UdIntms := SysTimeGetMs();
uiMsSecond := UDINT_TO_UINT((UdIntms - UdMsOffset)MOD 1000);   //计算微秒
DTimer_Str := UINT_TO_STRING(uiYear);
DTimer_Str := concat(DTimer_Str,'-');
DTimer_Str := concat(DTimer_Str,UINT_TO_STRING(uiMonth));
DTimer_Str := concat(DTimer_Str,'-');
DTimer_Str := concat(DTimer_Str,UINT_TO_STRING(uiDay));
DTimer_Str := concat(DTimer_Str,' ');
DTimer_Str := concat(DTimer_Str,UINT_TO_STRING(uiHour+8));
DTimer_Str := concat(DTimer_Str,':');
DTimer_Str := concat(DTimer_Str,UINT_TO_STRING(uiMinute));
DTimer_Str := concat(DTimer_Str,':');
DTimer_Str := concat(DTimer_Str,UINT_TO_STRING(uiSecond));
DTimer_Str := concat(DTimer_Str,':');
DTimer_Str := concat(DTimer_Str,UINT_TO_STRING(uiMsSecond));
DTimer_Str := concat(DTimer_Str,'    ');

log_Str := concat(Log_Data,'$R');
F_HANDL :=SysFileOpen(szFile:= Filename, am:=ACCESS_MODE.AM_APPEND, pResult:= ADR(F_err));  //打开文件
SysFileGetPos(hFile:= F_HANDL , pulPos:= ADR(F_pos));		//获取文件位置
SysFileSetPos(hFile:= F_HANDL, ulOffset:= F_pos);
SysFileWrite(hFile:=F_HANDL , pbyBuffer:= ADR(DTimer_Str) , ulSize:= SysStrLen(DTimer_Str) , pResult:= ADR(F_err));		// 写入时间
SysFileWrite(hFile:=F_HANDL , pbyBuffer:= ADR(log_Str) , ulSize:= SysStrLen(log_Str) , pResult:= ADR(F_err));		// 写入数据
SysFileClose(hFile:=F_HANDL );

Out_log := concat(DTimer_Str,log_Str);

END_FUNCTION_BLOCK

// Device/Application/modbus/getObjIndexC
FUNCTION_BLOCK FINAL getObjIndexC
VAR_INPUT
	iAdr	:UINT;
	iBit	:UINT;
END_VAR
VAR_OUTPUT
	iO1		:USINT;
	iO2		:USINT;
END_VAR
VAR
END_VAR

//已知指令地址，获取对应比例阀索引及油缸编号索引
CASE iAdr OF
	10,13:
		CASE iBit OF
			1:		iO1:=3;iO2:=1;//Q01-04
			2:		iO1:=4;iO2:=1;//Q05-08
			3:		iO1:=5;iO2:=1;//Q09-12
			4:		iO1:=6;iO2:=1;//Q13-14
			5:		iO1:=6;iO2:=2;//Q15
			6:		iO1:=7;iO2:=4;//Q17-21
			7:		iO1:=7;iO2:=5;//Q22-26
			8:		iO1:=1;iO2:=5;//Q28
			9:		iO1:=1;iO2:=4;//Q29-30
			ELSE	iO1:=0;iO2:=0;	
		END_CASE

	11,14:
		CASE iBit OF
			0:		iO1:=1;iO2:=3;//L00
			ELSE	iO1:=0;iO2:=0;
		END_CASE	
	
	12,15:
		CASE iBit OF
			0:		iO1:=1;iO2:=6;//L01
			1:		iO1:=2;iO2:=1;//L02-04
			2:		iO1:=2;iO2:=2;//L05
			3:		iO1:=2;iO2:=3;//L06-08
			4:		iO1:=2;iO2:=4;//L09
			5:		iO1:=2;iO2:=5;//L10-12
			6:		iO1:=6;iO2:=4;//L13
			7:		iO1:=6;iO2:=3;//L14-15
			8:		iO1:=6;iO2:=5;//L16
			9:		iO1:=7;iO2:=6;//L17
			10:		iO1:=7;iO2:=1;//L18-21
			11:		iO1:=7;iO2:=2;//L22
			12:		iO1:=7;iO2:=3;//L23-26
			13:		iO1:=7;iO2:=7;//L27
			14:		iO1:=1;iO2:=1;//L28
			15:		iO1:=1;iO2:=2;//L29-30
			ELSE	iO1:=0;iO2:=0;
		END_CASE	
	ELSE
		iO1:=0;iO2:=0;	
END_CASE

END_FUNCTION_BLOCK

// Device/Application/modbus/getColumnStr
FUNCTION_BLOCK FINAL getColumnStr
VAR_INPUT
	iI1		:UINT;
	iI2		:UINT;
END_VAR
VAR_OUTPUT
	strO	:STRING;
END_VAR
VAR
END_VAR

CASE iI1 OF
	1:
	CASE iI2 OF
		1:strO:='E28L1-E28L2';
		2:strO:='E29L-E30L';
		3:strO:='E00L';
		4:strO:='E29Q-E30Q';
		5:strO:='E28Q';
		6:strO:='E01L';
	END_CASE
	2:
	CASE iI2 OF
		1:strO:='E02L-E04L';
		2:strO:='E05L';
		3:strO:='E06L-E08L';
		4:strO:='E09L';
		5:strO:='E10L-E12L';
	END_CASE
	3:strO:='E01Q1-E04Q2';
	4:strO:='E05Q1-E08Q2';
	5:strO:='E09Q1-E12Q2';
	6:
	CASE iI2 OF
		1:strO:='E13Q-E14Q';
		2:strO:='E15Q';
		3:strO:='E14L-E15L';
		4:strO:='E13L';
		5:strO:='E16L1-E16L2';

	END_CASE
	7:
	CASE iI2 OF
		1:strO:='E18L-E21L';
		2:strO:='E22L';
		3:strO:='E23L-E26L';
		4:strO:='E17Q-E21Q';
		5:strO:='E22Q-E26Q';
		6:strO:='E17L1-E17L2';
		7:strO:='E27L1-E27L2';
	END_CASE	
END_CASE

END_FUNCTION_BLOCK

// Device/Application/modbus/getObjIndexE
FUNCTION_BLOCK getObjIndexE
VAR_INPUT
	iI1:INT;
	iI2:INT;
END_VAR
VAR_OUTPUT
	iAdr:USINT;
END_VAR
VAR
	
END_VAR

//Modbus中，输入油缸编号索引，返回用于地址用于写入伸出状态是否到位
CASE iI1 OF
	1:
		CASE iI2 OF
			1:iAdr:=139;//L28
			2:iAdr:=140;//L29-L30
			3:iAdr:=124;//L00
			4:iAdr:=119;//Q29-Q30
			5:iAdr:=118;//Q28
			6:iAdr:=125;//L01
		END_CASE
	2:
		CASE iI2 OF
			1:iAdr:=126;//L02-04
			2:iAdr:=127;//L05
			3:iAdr:=128;//L06-08
			4:iAdr:=129;//L09
			5:iAdr:=130;//L10-12
		END_CASE
	3:iAdr:=111;//Q01-04
	4:iAdr:=112;//Q05-08
	5:iAdr:=113;//Q09-12
	6:
		CASE iI2 OF
			1:iAdr:=114;//Q13-14
			2:iAdr:=115;//Q15
			3:iAdr:=132;//L14-15
			4:iAdr:=131;//L13
			5:iAdr:=133;//L16
		END_CASE
	7:
		CASE iI2 OF
			1:iAdr:=135;//L18-21
			2:iAdr:=136;//L22
			3:iAdr:=137;//L23-26
			4:iAdr:=116;//Q17-21
			5:iAdr:=117;//Q22-26
			6:iAdr:=134;//L17
			7:iAdr:=138;//L27
		END_CASE

ELSE	
	iAdr:=0;
END_CASE

END_FUNCTION_BLOCK

// Device/Application/modbus/getObjIndexR
FUNCTION_BLOCK getObjIndexR
VAR_INPUT
	iI1:INT;
	iI2:INT;
END_VAR
VAR_OUTPUT
	iAdr:USINT;
END_VAR
VAR
	
END_VAR

//Modbus中，输入油缸编号索引，返回用于地址用于写入缩回状态是否到位
CASE iI1 OF
	1:		
		CASE iI2 OF	
			1:iAdr:=170;//L28
			2:iAdr:=171;//L29-30
			3:iAdr:=155;//L00
			4:iAdr:=150;//Q29-30
			5:iAdr:=149;//Q28
			6:iAdr:=156;//L01
		END_CASE	
	2:		
		CASE iI2 OF	
			1:iAdr:=157;//L02-04
			2:iAdr:=158;//L05
			3:iAdr:=159;//L06-08
			4:iAdr:=160;//L09
			5:iAdr:=161;//L10-12
		END_CASE	
	3:iAdr:=142;//Q01-04		
	4:iAdr:=143;//Q05-08		
	5:iAdr:=144;//Q09-12		
	6:		
		CASE iI2 OF	
			1:iAdr:=145;//Q13-14
			2:iAdr:=146;//Q15
			3:iAdr:=163;//L14-15
			4:iAdr:=162;//L13
			5:iAdr:=164;//L16
		END_CASE	
	7:		
		CASE iI2 OF	
			1:iAdr:=166;//L18-21
			2:iAdr:=167;//L22
			3:iAdr:=168;//L23-26
			4:iAdr:=147;//Q17-21
			5:iAdr:=148;//Q22-26
			6:iAdr:=165;//L17
			7:iAdr:=169;//L27
		END_CASE	


ELSE	
	iAdr:=0;
END_CASE

END_FUNCTION_BLOCK

// Device/Application/rail_ceiling/positionRecord
PROGRAM positionRecord
VAR
	arrPosVal			:ARRAY[1..200] OF UINT;
	fbDatSav			:DatSave;
	iT1					:UINT;
	iT2					:UINT;
	iNum				:UINT;
END_VAR
VAR CONSTANT
	aOil	:ARRAY [1..7] OF UINT :=[9,11,8,8,8,8,23];		
END_VAR

iNum:=1;
FOR iT1:=1 TO 7 DO
	FOR iT2:=1 TO aOil[iT1] DO
		arrPosVal[iNum]:=REAL_TO_UINT(gImple.PV_GroupTi.arrPV[iT1].sNum[iT2].posVal.Current);
		iNum:=iNum+1;
	END_FOR
END_FOR
fbDatSav(Data_Arry:=arrPosVal , Num:= 75 , FilePath:= 'D:/DataSave', cycle:= T#7200S);

END_PROGRAM

// Device/Application/public_datum/datarecord/datSave
FUNCTION_BLOCK datSave
VAR_INPUT
	Data_Arry	: ARRAY[1..200] OF UINT;	// 数据输入 一次最大可以写入200个数据
	Num			: UINT;						// 存储数据个数
	FilePath 	: STRING := 'C:/DataSave'; 	// 存储文件夹
	cycle		: TIME;						// 更新一个文件夹时间
END_VAR
VAR_OUTPUT
END_VAR
VAR
	datetime	: DATE_AND_TIME;
	uiYear 		: UINT; 
    uiMonth 	: UINT; 
    uiDay 		: UINT; 
    uiHour 		: UINT; 
    uiMinute 	: UINT; 
    uiSecond 	: UINT;	
	uiMsSecond	: UINT;
	Last_S		: UINT:=100;
	UdMsOffset  : UDINT;
	UdIntms 	: UDINT;
	DTimer_Arry : ARRAY[1..7] OF UINT;
END_VAR
VAR
	File_Init	: BOOL :=TRUE;
	Frame_Cnt	: LINT;
	Data_Save_Init :BOOL:=TRUE;
	New_File_Ton: TON;
	Filename	: STRING;
	F_HANDL		: DWORD;
	F_err		: DWORD;
	F_pos		: DWORD;
END_VAR

datetime:=GetDateTime();   //获取时间
DTU.DTSplit(
		dtDateAndTime:= datetime, 
		puiYear:= ADR(uiYear), 
		puiMonth:=  ADR(uiMonth), 
		puiDay:=  ADR(uiDay), 
		puiHour:=  ADR(uiHour), 
		puiMinute:=  ADR(uiMinute), 
		puiSecond:= ADR(uiSecond) );

IF  Data_Save_Init THEN			//数据存储初始化
	IF uiSecond = Last_S +1 OR  uiSecond = Last_S -59 THEN
		UdMsOffset := SysTimeGetMs();
		Last_S :=  uiSecond;
	ELSE
		Last_S :=  uiSecond;
		RETURN;
	END_IF
    Data_Save_Init := FALSE;
END_IF

IF 	File_Init  THEN          //创建文件
	Filename := FilePath;
	Filename := concat(Filename,'/');
	Filename := concat(Filename,UINT_TO_STRING(uiYear));
	Filename := concat(Filename,'_');
	Filename := concat(Filename,UINT_TO_STRING(uiMonth));
	Filename := concat(Filename,'_');
	Filename := concat(Filename,UINT_TO_STRING(uiDay));
	Filename := concat(Filename,'_');
	Filename := concat(Filename,UINT_TO_STRING(uiHour+8));
 	Filename := concat(Filename,'_');
	Filename := concat(Filename,UINT_TO_STRING(uiMinute));
	Filename := concat(Filename,'_');
	Filename := concat(Filename,UINT_TO_STRING(uiSecond));
    Filename := concat(Filename,'_Data.bin');
	Frame_Cnt := 0;
	F_HANDL :=SysFileOpen(szFile:= Filename, am:=ACCESS_MODE.AM_WRITE, pResult:= ADR(F_err));  //创建新文件
	SysFileClose(hFile:=F_HANDL );
	File_Init := FALSE;
	New_File_Ton(IN:= FALSE , PT:= cycle, Q=> , ET=> );  //复位
END_IF

New_File_Ton(IN:= TRUE , PT:= cycle, Q=> , ET=> );			//4小时创建一个新文件
IF New_File_Ton.Q THEN
	File_Init := TRUE;	
END_IF



UdIntms := SysTimeGetMs();
DTimer_Arry[1] := uiYear;
DTimer_Arry[2] := uiMonth;
DTimer_Arry[3] := uiDay;
DTimer_Arry[4] := uiHour+8;
DTimer_Arry[5] := uiMinute;
DTimer_Arry[6] := uiSecond;
DTimer_Arry[7] := UDINT_TO_UINT((UdIntms - UdMsOffset)MOD 1000);

Frame_Cnt := Frame_Cnt + 1;    	//帧计数增加

F_HANDL :=SysFileOpen(szFile:= Filename, am:=ACCESS_MODE.AM_APPEND, pResult:= ADR(F_err));  //打开文件
SysFileGetPos(hFile:= F_HANDL , pulPos:= ADR(F_pos));		//获取文件位置
SysFileSetPos(hFile:= F_HANDL, ulOffset:= 0);	//设置帧位置
SysFileWrite(hFile:=F_HANDL , pbyBuffer:= ADR(Frame_Cnt) , ulSize:= SIZEOF(Frame_Cnt) , pResult:= ADR(F_err));    //修改总帧数
IF F_pos <> 0 THEN		//不是新文件，设置写入位置
	SysFileSetPos(hFile:= F_HANDL, ulOffset:= F_pos);
END_IF
SysFileWrite(hFile:=F_HANDL , pbyBuffer:= ADR(DTimer_Arry) , ulSize:= SIZEOF(DTimer_Arry) , pResult:= ADR(F_err));  // 保存时间
SysFileWrite(hFile:=F_HANDL , pbyBuffer:= ADR(Data_Arry) , ulSize:= SIZEOF(UINT)*Num , pResult:= ADR(F_err));		// 保存数据
SysFileClose(hFile:=F_HANDL );

END_FUNCTION_BLOCK

// Device/Application/can/canRx
PROGRAM canRx
VAR
		T_CNT   :UINT;
END_VAR

T_CNT := T_CNT+1;
IF  T_CNT > 1000 THEN
	 T_CNT := 1;
END_IF


swmc_C05_Rx(T_CNT,ADR(gImple.hydraPresStation),ADR(gImple.PV_GroupTi));
swmc_C06_Rx(T_CNT,ADR(gImple.hydraPresStation),ADR(gImple.PV_GroupTi));
swmc_C12_Rx(T_CNT,ADR(gImple.PV_GroupTi));

END_PROGRAM

// Device/Application/can/swmc_C05_Rx
FUNCTION swmc_C05_Rx : BOOL
VAR_INPUT
	CNT				: UINT;
	psYyz			: POINTER TO YyStation;
	psPVTi			: POINTER TO propValveModule_Ti;

END_VAR
VAR
	frame	 	    : Can_baseframe;
	COB_ID			: UINT;
	I				: UINT;
	Pre				: UINT;
	pos				: WORD;
END_VAR

IF gCan.C5RxMsg.RxCounter <>  gCan.C5RxCounter THEN    //接收到新的数据

	FOR  I := 1 TO  gCan.C5RxMsg.NoOfRxMessages DO
		frame :=CAN_Read_Data_SWMC(5,I);
		COB_ID :=	frame.id;    //获取ID
		CASE COB_ID OF     //根据ID解析协议
		
		//C5-0x350
			16#350://接收C5送来的数据
				pos := BYTE_TO_WORD(frame.data[1]) OR SHL(BYTE_TO_WORD(frame.data[2]),8);  	
				psPVTi^.arrPV[3].sNum[1].posVal.Current:= pos*0.1;
				pos := BYTE_TO_WORD(frame.data[3]) OR SHL(BYTE_TO_WORD(frame.data[4]),8);  
				psPVTi^.arrPV[3].sNum[2].posVal.Current:= pos*0.1;	
				pos := BYTE_TO_WORD(frame.data[5]) OR SHL(BYTE_TO_WORD(frame.data[6]),8);  
				psPVTi^.arrPV[3].sNum[3].posVal.Current:= pos*0.1;	
				pos := BYTE_TO_WORD(frame.data[7]) OR SHL(BYTE_TO_WORD(frame.data[8]),8);  	
				psPVTi^.arrPV[3].sNum[4].posVal.Current:= pos*0.1;
			
			//C5-0x351
			16#351://接收C5送来的数据
				pos := BYTE_TO_WORD(frame.data[1]) OR SHL(BYTE_TO_WORD(frame.data[2]),8);  	
				psPVTi^.arrPV[3].sNum[5].posVal.Current:= pos*0.1;	
				pos := BYTE_TO_WORD(frame.data[3]) OR SHL(BYTE_TO_WORD(frame.data[4]),8);  	
				psPVTi^.arrPV[3].sNum[6].posVal.Current:= pos*0.1;	
				pos := BYTE_TO_WORD(frame.data[5]) OR SHL(BYTE_TO_WORD(frame.data[6]),8);  	
				psPVTi^.arrPV[3].sNum[7].posVal.Current:= pos*0.1;	
				pos := BYTE_TO_WORD(frame.data[7]) OR SHL(BYTE_TO_WORD(frame.data[8]),8);  	
				psPVTi^.arrPV[3].sNum[8].posVal.Current:= pos*0.1;
			
			//C5-0x352
			16#352://接收C5送来的数据
			pos := BYTE_TO_WORD(frame.data[1]) OR SHL(BYTE_TO_WORD(frame.data[2]),8);  	
				psPVTi^.arrPV[4].sNum[1].posVal.Current:= pos*0.1;	
				pos := BYTE_TO_WORD(frame.data[3]) OR SHL(BYTE_TO_WORD(frame.data[4]),8);  	
				psPVTi^.arrPV[4].sNum[2].posVal.Current:= pos*0.1;		
				pos := BYTE_TO_WORD(frame.data[5]) OR SHL(BYTE_TO_WORD(frame.data[6]),8);  	
				psPVTi^.arrPV[4].sNum[3].posVal.Current:= pos*0.1;		
				pos := BYTE_TO_WORD(frame.data[7]) OR SHL(BYTE_TO_WORD(frame.data[8]),8);  	
				psPVTi^.arrPV[4].sNum[4].posVal.Current:= pos*0.1;	
			
			//C5-0x353
			16#353://接收C5送来的数据
				pos := BYTE_TO_WORD(frame.data[1]) OR SHL(BYTE_TO_WORD(frame.data[2]),8);  	
				psPVTi^.arrPV[4].sNum[5].posVal.Current:= pos*0.1;		
				pos := BYTE_TO_WORD(frame.data[3]) OR SHL(BYTE_TO_WORD(frame.data[4]),8);  	
				psPVTi^.arrPV[4].sNum[6].posVal.Current:= pos*0.1;		
				pos := BYTE_TO_WORD(frame.data[5]) OR SHL(BYTE_TO_WORD(frame.data[6]),8);  	
				psPVTi^.arrPV[4].sNum[7].posVal.Current:= pos*0.1;		
				pos := BYTE_TO_WORD(frame.data[7]) OR SHL(BYTE_TO_WORD(frame.data[8]),8);  	
				psPVTi^.arrPV[4].sNum[8].posVal.Current:= pos*0.1;	
			
			//C5-0x354
			16#354://接收C5送来的数据
			pos := BYTE_TO_WORD(frame.data[1]) OR SHL(BYTE_TO_WORD(frame.data[2]),8);  	
				psPVTi^.arrPV[5].sNum[1].posVal.Current:= pos*0.1;		
				pos := BYTE_TO_WORD(frame.data[3]) OR SHL(BYTE_TO_WORD(frame.data[4]),8);  	
				psPVTi^.arrPV[5].sNum[2].posVal.Current:= pos*0.1;		
				pos := BYTE_TO_WORD(frame.data[5]) OR SHL(BYTE_TO_WORD(frame.data[6]),8);  	
				psPVTi^.arrPV[5].sNum[3].posVal.Current:= pos*0.1;		
				pos := BYTE_TO_WORD(frame.data[7]) OR SHL(BYTE_TO_WORD(frame.data[8]),8);  	
				psPVTi^.arrPV[5].sNum[4].posVal.Current:= pos*0.1;	
			
			//C5-0x355
			16#355://接收C5送来的数据
			pos := BYTE_TO_WORD(frame.data[1]) OR SHL(BYTE_TO_WORD(frame.data[2]),8);  	
				psPVTi^.arrPV[5].sNum[5].posVal.Current:= pos*0.1;		
				pos := BYTE_TO_WORD(frame.data[3]) OR SHL(BYTE_TO_WORD(frame.data[4]),8);  	
				psPVTi^.arrPV[5].sNum[6].posVal.Current:= pos*0.1;		
				pos := BYTE_TO_WORD(frame.data[5]) OR SHL(BYTE_TO_WORD(frame.data[6]),8);  	
				psPVTi^.arrPV[5].sNum[7].posVal.Current:= pos*0.1;		
				pos := BYTE_TO_WORD(frame.data[7]) OR SHL(BYTE_TO_WORD(frame.data[8]),8);  	
				psPVTi^.arrPV[5].sNum[8].posVal.Current:= pos*0.1;	
			

	
			//C5-0x356
			16#356:           //接收C5送来的数据
			(*
				Pre :=BYTE_TO_WORD(frame.data[1]) OR SHL(BYTE_TO_WORD(frame.data[2]),8);
				psYyz^.Status.pressureV10:= 	(Pre-4000)/16000.0*400;	
				Pre :=BYTE_TO_WORD(frame.data[3]) OR SHL(BYTE_TO_WORD(frame.data[4]),8);
				psYyz^.Status.pressureV11:= 	(Pre-4000)/16000.0*400;	
			*)
			
	
		END_CASE
	END_FOR
	gCan.C5RxCounter := gCan.C5RxMsg.RxCounter ;
END_IF

END_FUNCTION

// Device/Application/can/CAN_Read_Data_SWMC
FUNCTION CAN_Read_Data_SWMC : Can_baseframe
VAR_INPUT
	SWMC_ID	 :UINT;		//接收SWMC控制ID
	I	 	 :UINT;      //接收缓冲区域
END_VAR
VAR
	frame :Can_baseframe;
END_VAR

CASE  SWMC_ID OF

	5:                       //SWMC-C5
		frame.id 	:= (gCan.C5RxMsg.RXMsg[I].RxMsg_CobId-8)/32;
		frame.data 	:= gCan.C5RxMsg.RXMsg[I].RxMsg_Byte;
				
	6:                       //SWMC-C6
		frame.id 	:= (gCan.C6RxMsg.RXMsg[I].RxMsg_CobId-8)/32;
		frame.data 	:= gCan.C6RxMsg.RXMsg[I].RxMsg_Byte;

	12:						//SWMC-C12
		frame.id 	:= (gCan.C12RxMsg.RXMsg[I].RxMsg_CobId-8)/32;
		frame.data 	:= gCan.C12RxMsg.RXMsg[I].RxMsg_Byte;	
		
	ELSE				//Other
		frame.id := 0;
		frame.data[1] := 0;
		frame.data[2] := 0;
		frame.data[3] := 0;
		frame.data[4] := 0;
		frame.data[5] := 0;
		frame.data[6] := 0;
		frame.data[7] := 0;
		frame.data[8] := 0;
END_CASE
Can_Read_data_SWMC := frame;

END_FUNCTION

// Device/Application/can/swmc_C06_Rx
FUNCTION swmc_C06_Rx : BOOL
VAR_INPUT
	CNT				: UINT;
	psYyz			: POINTER TO YyStation;
	psPVTi			: POINTER TO propValveModule_Ti;

END_VAR
VAR
	frame	 	    : Can_baseframe;
	COB_ID			: UINT;
	I				: UINT;
	Pre				: UINT;
	pos				: WORD;
END_VAR

IF gCan.C6RxMsg.RxCounter <>  gCan.C6RxCounter THEN    //接收到新的数据

	FOR  I := 1 TO  gCan.C6RxMsg.NoOfRxMessages DO
		frame :=CAN_Read_Data_SWMC(6,I);
		COB_ID :=	frame.id;    //获取ID
		CASE COB_ID OF     //根据ID解析协议
	
		
			//C6-0x360
			16#360:           //接收C6送来的数据
				pos:=BYTE_TO_WORD(frame.data[1]) OR SHL(BYTE_TO_WORD(frame.data[2]),8);
				psPVTi^.arrPV[1].sNum[3].posVal.Current:=pos*0.1;
				pos:=BYTE_TO_WORD(frame.data[3]) OR SHL(BYTE_TO_WORD(frame.data[4]),8);
				psPVTi^.arrPV[1].sNum[4].posVal.Current:=pos*0.1;
				pos:=BYTE_TO_WORD(frame.data[5]) OR SHL(BYTE_TO_WORD(frame.data[6]),8);
				psPVTi^.arrPV[1].sNum[9].posVal.Current:=pos*0.1;
				pos:=BYTE_TO_WORD(frame.data[7]) OR SHL(BYTE_TO_WORD(frame.data[8]),8);
				psPVTi^.arrPV[1].sNum[5].posVal.Current:=pos*0.1;
			

			//C6-0x361
			16#361:           //接收C6送来的数据
				pos:=BYTE_TO_WORD(frame.data[1]) OR SHL(BYTE_TO_WORD(frame.data[2]),8);
				psPVTi^.arrPV[1].sNum[8].posVal.Current:=pos*0.1;
				pos:=BYTE_TO_WORD(frame.data[3]) OR SHL(BYTE_TO_WORD(frame.data[4]),8);
				psPVTi^.arrPV[1].sNum[6].posVal.Current:=pos*0.1;
				pos:=BYTE_TO_WORD(frame.data[5]) OR SHL(BYTE_TO_WORD(frame.data[6]),8);
				psPVTi^.arrPV[1].sNum[7].posVal.Current:=pos*0.1;
				pos:=BYTE_TO_WORD(frame.data[7]) OR SHL(BYTE_TO_WORD(frame.data[8]),8);
				psPVTi^.arrPV[2].sNum[1].posVal.Current:=pos*0.1;
			//C6-0x362
			16#362:           //接收C6送来的数据
				pos:=BYTE_TO_WORD(frame.data[1]) OR SHL(BYTE_TO_WORD(frame.data[2]),8);
				psPVTi^.arrPV[2].sNum[2].posVal.Current:=pos*0.1;
				pos:=BYTE_TO_WORD(frame.data[3]) OR SHL(BYTE_TO_WORD(frame.data[4]),8);
				psPVTi^.arrPV[2].sNum[3].posVal.Current:=pos*0.1;
				pos:=BYTE_TO_WORD(frame.data[5]) OR SHL(BYTE_TO_WORD(frame.data[6]),8);
				psPVTi^.arrPV[2].sNum[4].posVal.Current:=pos*0.1;
				pos:=BYTE_TO_WORD(frame.data[7]) OR SHL(BYTE_TO_WORD(frame.data[8]),8);
				psPVTi^.arrPV[2].sNum[5].posVal.Current:=pos*0.1;
			//C6-0x363
			16#363:           //接收C6送来的数据
				pos:=BYTE_TO_WORD(frame.data[1]) OR SHL(BYTE_TO_WORD(frame.data[2]),8);
				psPVTi^.arrPV[2].sNum[6].posVal.Current:=pos*0.1;
				pos:=BYTE_TO_WORD(frame.data[3]) OR SHL(BYTE_TO_WORD(frame.data[4]),8);
				psPVTi^.arrPV[2].sNum[7].posVal.Current:=pos*0.1;
				pos:=BYTE_TO_WORD(frame.data[5]) OR SHL(BYTE_TO_WORD(frame.data[6]),8);
				psPVTi^.arrPV[2].sNum[8].posVal.Current:=pos*0.1;
				pos:=BYTE_TO_WORD(frame.data[7]) OR SHL(BYTE_TO_WORD(frame.data[8]),8);
				psPVTi^.arrPV[2].sNum[9].posVal.Current:=pos*0.1;
			//C6-0x364
			16#364:           //接收C6送来的数据
				pos:=BYTE_TO_WORD(frame.data[1]) OR SHL(BYTE_TO_WORD(frame.data[2]),8);
				psPVTi^.arrPV[2].sNum[10].posVal.Current:=pos*0.1;
				pos:=BYTE_TO_WORD(frame.data[3]) OR SHL(BYTE_TO_WORD(frame.data[4]),8);
				psPVTi^.arrPV[2].sNum[11].posVal.Current:=pos*0.1;
				pos:=BYTE_TO_WORD(frame.data[5]) OR SHL(BYTE_TO_WORD(frame.data[6]),8);
				psPVTi^.arrPV[6].sNum[6].posVal.Current:=pos*0.1;
				pos:=BYTE_TO_WORD(frame.data[7]) OR SHL(BYTE_TO_WORD(frame.data[8]),8);
				psPVTi^.arrPV[6].sNum[4].posVal.Current:=pos*0.1;
			//C6-0x365
			16#365:           //接收C6送来的数据
				pos:=BYTE_TO_WORD(frame.data[1]) OR SHL(BYTE_TO_WORD(frame.data[2]),8);
				psPVTi^.arrPV[6].sNum[5].posVal.Current:=pos*0.1;
				pos:=BYTE_TO_WORD(frame.data[3]) OR SHL(BYTE_TO_WORD(frame.data[4]),8);
				psPVTi^.arrPV[6].sNum[1].posVal.Current:=pos*0.1;
				pos:=BYTE_TO_WORD(frame.data[5]) OR SHL(BYTE_TO_WORD(frame.data[6]),8);
				psPVTi^.arrPV[6].sNum[2].posVal.Current:=pos*0.1;
				pos:=BYTE_TO_WORD(frame.data[7]) OR SHL(BYTE_TO_WORD(frame.data[8]),8);
				psPVTi^.arrPV[6].sNum[3].posVal.Current:=pos*0.1;
				
		
			//C6-0x366
			16#366:           //接收C6送来的数据
				//Pre :=BYTE_TO_WORD(frame.data[1]) OR SHL(BYTE_TO_WORD(frame.data[2]),8);
	 			//psYyz^.Status.pressureV8:= 	(Pre-4000)/16000.0*400;	
				//Pre :=BYTE_TO_WORD(frame.data[3]) OR SHL(BYTE_TO_WORD(frame.data[4]),8);
	 			//psYyz^.Status.pressureV9:= 	(Pre-4000)/16000.0*400;	
				pos	:=BYTE_TO_WORD(frame.data[5]) OR SHL(BYTE_TO_WORD(frame.data[6]),8);
				psPVTi^.arrAddtion[1].sPlateStatus.sSensor.Current:=pos*0.1;
				pos	:=BYTE_TO_WORD(frame.data[7]) OR SHL(BYTE_TO_WORD(frame.data[8]),8);
				psPVTi^.arrAddtion[2].sPlateStatus.sSensor.Current:=pos*0.1;
				
		END_CASE
	END_FOR
	gCan.C6RxCounter := gCan.C6RxMsg.RxCounter ;
END_IF

END_FUNCTION

// Device/Application/can/swmc_C12_Rx
FUNCTION swmc_C12_Rx : BOOL
VAR_INPUT
	CNT				: UINT;
	psPVTi			: POINTER TO propValveModule_Ti;
END_VAR
VAR
	frame	 	    : Can_baseframe;
	COB_ID			: UINT;
	I				: UINT;
	Pre				: UINT;
	pos				: WORD;
END_VAR

IF gCan.C12RxMsg.RxCounter <>  gCan.C12RxCounter THEN    //接收到新的数据

	FOR  I := 1 TO  gCan.C12RxMsg.NoOfRxMessages DO
		frame :=CAN_Read_Data_SWMC(12,I);
		COB_ID :=	frame.id;    //获取ID
		CASE COB_ID OF     //根据ID解析协议
		
		
			//C12-0x3C0
			16#3C0:           //接收C12送来的数据
				pos := BYTE_TO_WORD(frame.data[ 1 ]) OR SHL(BYTE_TO_WORD(frame.data[ 2 ]),8);  	
				psPVTi^.arrPV[ 6 ].sNum[ 7 ].posVal.Current:= pos*0.1;	
				pos := BYTE_TO_WORD(frame.data[ 3 ]) OR SHL(BYTE_TO_WORD(frame.data[ 4 ]),8);  
				psPVTi^.arrPV[ 6 ].sNum[ 8 ].posVal.Current:= pos*0.1;		
				pos := BYTE_TO_WORD(frame.data[ 5 ]) OR SHL(BYTE_TO_WORD(frame.data[ 6 ]),8);  
				psPVTi^.arrPV[ 7 ].sNum[ 20 ].posVal.Current:= pos*0.1;	
				pos := BYTE_TO_WORD(frame.data[ 7 ]) OR SHL(BYTE_TO_WORD(frame.data[ 8 ]),8);  	
				psPVTi^.arrPV[ 7 ].sNum[ 21 ].posVal.Current:= pos*0.1;

			//C6-0x3C1
			16#3C1:           //接收C12送来的数据
				pos := BYTE_TO_WORD(frame.data[ 1 ]) OR SHL(BYTE_TO_WORD(frame.data[ 2 ]),8);  	
				psPVTi^.arrPV[ 7 ].sNum[ 1 ].posVal.Current:= pos*0.1;	
				pos := BYTE_TO_WORD(frame.data[ 3 ]) OR SHL(BYTE_TO_WORD(frame.data[ 4 ]),8);  	
				psPVTi^.arrPV[ 7 ].sNum[ 2 ].posVal.Current:= pos*0.1;	
				pos := BYTE_TO_WORD(frame.data[ 5 ]) OR SHL(BYTE_TO_WORD(frame.data[ 6 ]),8);  	
				psPVTi^.arrPV[ 7 ].sNum[ 3 ].posVal.Current:= pos*0.1;	
				pos := BYTE_TO_WORD(frame.data[ 7 ]) OR SHL(BYTE_TO_WORD(frame.data[ 8 ]),8);  	
				psPVTi^.arrPV[ 7 ].sNum[ 4 ].posVal.Current:= pos*0.1;
			//C6-0x3C2
			16#3C2:           //接收C12送来的数据
				pos := BYTE_TO_WORD(frame.data[ 1 ]) OR SHL(BYTE_TO_WORD(frame.data[ 2 ]),8);  	
				psPVTi^.arrPV[ 7 ].sNum[ 5 ].posVal.Current:= pos*0.1;	
				pos := BYTE_TO_WORD(frame.data[ 3 ]) OR SHL(BYTE_TO_WORD(frame.data[ 4 ]),8);  	
				psPVTi^.arrPV[ 7 ].sNum[ 6 ].posVal.Current:= pos*0.1;		
				pos := BYTE_TO_WORD(frame.data[ 5 ]) OR SHL(BYTE_TO_WORD(frame.data[ 6 ]),8);  	
				psPVTi^.arrPV[ 7 ].sNum[ 7 ].posVal.Current:= pos*0.1;		
				pos := BYTE_TO_WORD(frame.data[ 7 ]) OR SHL(BYTE_TO_WORD(frame.data[ 8 ]),8);  	
				psPVTi^.arrPV[ 7 ].sNum[ 8 ].posVal.Current:= pos*0.1;	
			//C6-0x3C3
			16#3C3:           //接收C12送来的数据
				pos := BYTE_TO_WORD(frame.data[ 1 ]) OR SHL(BYTE_TO_WORD(frame.data[ 2 ]),8);  	
				psPVTi^.arrPV[ 7 ].sNum[ 9 ].posVal.Current:= pos*0.1;		
				pos := BYTE_TO_WORD(frame.data[ 3 ]) OR SHL(BYTE_TO_WORD(frame.data[ 4 ]),8);  	
				psPVTi^.arrPV[ 7 ].sNum[ 22 ].posVal.Current:= pos*0.1;		
				pos := BYTE_TO_WORD(frame.data[ 5 ]) OR SHL(BYTE_TO_WORD(frame.data[ 6 ]),8);  	
				psPVTi^.arrPV[7 ].sNum[ 23 ].posVal.Current:= pos*0.1;		
				pos := BYTE_TO_WORD(frame.data[ 7 ]) OR SHL(BYTE_TO_WORD(frame.data[ 8 ]),8);  	
				psPVTi^.arrPV[ 1 ].sNum[ 1 ].posVal.Current:= pos*0.1;	
			//C6-0x3C4
			16#3C4:           //接收C12送来的数据
				pos := BYTE_TO_WORD(frame.data[ 1 ]) OR SHL(BYTE_TO_WORD(frame.data[ 2 ]),8);  	
				psPVTi^.arrPV[ 1 ].sNum[ 2 ].posVal.Current:= pos*0.1;		
				pos := BYTE_TO_WORD(frame.data[ 3 ]) OR SHL(BYTE_TO_WORD(frame.data[ 4 ]),8);  	
				psPVTi^.arrPV[ 7 ].sNum[ 10 ].posVal.Current:= pos*0.1;		
				pos := BYTE_TO_WORD(frame.data[ 5 ]) OR SHL(BYTE_TO_WORD(frame.data[ 6 ]),8);  	
				psPVTi^.arrPV[ 7 ].sNum[ 11 ].posVal.Current:= pos*0.1;		
				pos := BYTE_TO_WORD(frame.data[ 7 ]) OR SHL(BYTE_TO_WORD(frame.data[ 8 ]),8);  	
				psPVTi^.arrPV[7 ].sNum[ 12 ].posVal.Current:= pos*0.1;	
			//C6-0x3C5
			16#3C5:           //接收C12送来的数据
				pos := BYTE_TO_WORD(frame.data[ 1 ]) OR SHL(BYTE_TO_WORD(frame.data[ 2 ]),8);  	
				psPVTi^.arrPV[ 7 ].sNum[ 13 ].posVal.Current:= pos*0.1;		
				pos := BYTE_TO_WORD(frame.data[ 3 ]) OR SHL(BYTE_TO_WORD(frame.data[ 4 ]),8);  	
				psPVTi^.arrPV[ 7 ].sNum[ 14 ].posVal.Current:= pos*0.1;		
				pos := BYTE_TO_WORD(frame.data[ 5 ]) OR SHL(BYTE_TO_WORD(frame.data[ 6 ]),8);  	
				psPVTi^.arrPV[ 7 ].sNum[ 15 ].posVal.Current:= pos*0.1;		
				pos := BYTE_TO_WORD(frame.data[ 7 ]) OR SHL(BYTE_TO_WORD(frame.data[ 8 ]),8);  	
				psPVTi^.arrPV[ 7 ].sNum[ 16 ].posVal.Current:= pos*0.1;
			//C6-0x3C6
			16#3C6:           //接收C12送来的数据
				pos := BYTE_TO_WORD(frame.data[ 1 ]) OR SHL(BYTE_TO_WORD(frame.data[ 2 ]),8);  	
				psPVTi^.arrPV[ 7 ].sNum[ 17 ].posVal.Current:= pos*0.1;		
				pos := BYTE_TO_WORD(frame.data[ 3 ]) OR SHL(BYTE_TO_WORD(frame.data[ 4 ]),8);  	
				psPVTi^.arrPV[ 7 ].sNum[ 18 ].posVal.Current:= pos*0.1;		
				pos := BYTE_TO_WORD(frame.data[ 5 ]) OR SHL(BYTE_TO_WORD(frame.data[ 6 ]),8);  	
				psPVTi^.arrPV[ 7 ].sNum[ 19 ].posVal.Current:= pos*0.1;		
						
		
			
		END_CASE
	END_FOR
	gCan.C12RxCounter := gCan.C12RxMsg.RxCounter ;
END_IF

END_FUNCTION

// Device/Application/public_datum/otherContent/rail_floor/floorRailAct
PROGRAM floorRailAct
VAR
	bInitialize		:BOOL:=TRUE;
	iVD				:INT;
	iVD1			:INT;
END_VAR
VAR CONSTANT
	aNo		:ARRAY [1..7] OF INT :=[ 7, 5,1,1,1,5, 7];		//每个比例阀下开关阀的数量(天轨):arrMappingRealNumTiG
	aOil	:ARRAY [1..7] OF INT :=[12,11,8,8,8,8,23];		
END_VAR

IF bInitialize THEN	//初始化
	floorRailAct.initName();
	floorRailAct.initRange();
	bInitialize:=FALSE;
END_IF
statusDisplayDi();
CommandDeliverDi();

ACTION statusDisplayDi:
//初始化：名称显示，油缸位移范围赋值
initName();
initRange();


//	gUI.界面值<--gImple.传感器位置值;

//比例阀DTD1
FOR iVD	:=1 TO 12 DO
	gUI.DiG.arrPV[1].sNum[iVD].rPosition:=gImple.PV_GroupDi.arrPV[1].sNum[iVD].posVal.Current;
	gUI.DiG.arrPV[1].sNum[iVD].rPercent:=statusPercentCalcDi(ADR(gImple.PV_GroupDi),1,iVD);
	gUI.DiG.arrPV[1].sNum[iVD].strName:=gUI.DiG_NameInit.strName[1,iVD];
END_FOR

//比例阀DTD2
FOR iVD	:=1 TO 11 DO
	gUI.DiG.arrPV[2].sNum[iVD].rPosition:=gImple.PV_GroupDi.arrPV[2].sNum[iVD].posVal.Current;
	gUI.DiG.arrPV[2].sNum[iVD].rPercent:=statusPercentCalcDi(ADR(gImple.PV_GroupDi),2,iVD);
	gUI.DiG.arrPV[2].sNum[iVD].strName:=gUI.DiG_NameInit.strName[2,iVD];
END_FOR

//比例阀DTD345
FOR iVD	:=1 TO 8 DO

	gUI.DiG.arrPV[3].sNum[iVD].rPosition:=gImple.PV_GroupDi.arrPV[3].sNum[iVD].posVal.Current;
	gUI.DiG.arrPV[4].sNum[iVD].rPosition:=gImple.PV_GroupDi.arrPV[4].sNum[iVD].posVal.Current;
	gUI.DiG.arrPV[5].sNum[iVD].rPosition:=gImple.PV_GroupDi.arrPV[5].sNum[iVD].posVal.Current;
	
	gUI.DiG.arrPV[3].sNum[iVD].rPercent:=statusPercentCalcDi(ADR(gImple.PV_GroupDi),3,iVD);
	gUI.DiG.arrPV[4].sNum[iVD].rPercent:=statusPercentCalcDi(ADR(gImple.PV_GroupDi),4,iVD);
	gUI.DiG.arrPV[5].sNum[iVD].rPercent:=statusPercentCalcDi(ADR(gImple.PV_GroupDi),5,iVD);
	
	gUI.DiG.arrPV[3].sNum[iVD].strName:=gUI.DiG_NameInit.strName[3,iVD];
	gUI.DiG.arrPV[4].sNum[iVD].strName:=gUI.DiG_NameInit.strName[4,iVD];
	gUI.DiG.arrPV[5].sNum[iVD].strName:=gUI.DiG_NameInit.strName[5,iVD];
END_FOR

//比例阀DTD6
FOR iVD	:=1 TO 8 DO
	gUI.DiG.arrPV[6].sNum[iVD].rPosition:=gImple.PV_GroupDi.arrPV[6].sNum[iVD].posVal.Current;
	gUI.DiG.arrPV[6].sNum[iVD].rPercent:=statusPercentCalcDi(ADR(gImple.PV_GroupDi),6,iVD);
	gUI.DiG.arrPV[6].sNum[iVD].strName:=gUI.DiG_NameInit.strName[6,iVD];
END_FOR

//比例阀DTD7
FOR iVD	:=1 TO 23 DO
	gUI.DiG.arrPV[7].sNum[iVD].rPosition:=gImple.PV_GroupDi.arrPV[7].sNum[iVD].posVal.Current;
	gUI.DiG.arrPV[7].sNum[iVD].rPercent:=statusPercentCalcDi(ADR(gImple.PV_GroupDi),7,iVD);
	gUI.DiG.arrPV[7].sNum[iVD].strName:=gUI.DiG_NameInit.strName[7,iVD];
END_FOR




//percentBar
(*
gUI.DiG1.D00Q1.rPercent	:=

*)
END_ACTION

METHOD CommandDeliverDi : BOOL
VAR_INPUT
	
END_VAR
END_METHOD

ACTION initName:
gUI.DiG_NameInit.strName[1,1]	:=	'D00Q1'	;
gUI.DiG_NameInit.strName[1,2]	:=	'D00Q2'	;
gUI.DiG_NameInit.strName[1,3]	:=	'D28L1'	;
gUI.DiG_NameInit.strName[1,4]	:=	'D28L2'	;
gUI.DiG_NameInit.strName[1,5]	:=	'D29L'	;
gUI.DiG_NameInit.strName[1,6]	:=	'D30L'	;
gUI.DiG_NameInit.strName[1,7]	:=	'D00L1'	;
gUI.DiG_NameInit.strName[1,8]	:=	'D00L2'	;
gUI.DiG_NameInit.strName[1,9]	:=	'D01L'	;
gUI.DiG_NameInit.strName[1,10]	:=	'D28Q'	;
gUI.DiG_NameInit.strName[1,11]	:=	'D29Q'	;
gUI.DiG_NameInit.strName[1,12]	:=	'D30Q'	;

gUI.DiG_NameInit.strName[2,1]	:=	'D02L'	;
gUI.DiG_NameInit.strName[2,2]	:=	'D03L'	;
gUI.DiG_NameInit.strName[2,3]	:=	'D04L'	;
gUI.DiG_NameInit.strName[2,4]	:=	'D05L'	;
gUI.DiG_NameInit.strName[2,5]	:=	'D06L'	;
gUI.DiG_NameInit.strName[2,6]	:=	'D07L'	;
gUI.DiG_NameInit.strName[2,7]	:=	'D08L'	;
gUI.DiG_NameInit.strName[2,8]	:=	'D09L'	;
gUI.DiG_NameInit.strName[2,9]	:=	'D10L'	;
gUI.DiG_NameInit.strName[2,10]	:=	'D11L'	;
gUI.DiG_NameInit.strName[2,11]	:=	'D12L'	;
	
gUI.DiG_NameInit.strName[3,1]	:=	'D01Q1'	;
gUI.DiG_NameInit.strName[3,2]	:=	'D01Q2'	;
gUI.DiG_NameInit.strName[3,3]	:=	'D02Q1'	;
gUI.DiG_NameInit.strName[3,4]	:=	'D02Q2'	;
gUI.DiG_NameInit.strName[3,5]	:=	'D03Q1'	;
gUI.DiG_NameInit.strName[3,6]	:=	'D03Q2'	;
gUI.DiG_NameInit.strName[3,7]	:=	'D04Q1'	;
gUI.DiG_NameInit.strName[3,8]	:=	'D04Q2'	;
gUI.DiG_NameInit.strName[4,1]	:=	'D05Q1'	;
gUI.DiG_NameInit.strName[4,2]	:=	'D05Q2'	;
gUI.DiG_NameInit.strName[4,3]	:=	'D06Q1'	;
gUI.DiG_NameInit.strName[4,4]	:=	'D06Q2'	;
gUI.DiG_NameInit.strName[4,5]	:=	'D07Q1'	;
gUI.DiG_NameInit.strName[4,6]	:=	'D07Q2'	;
gUI.DiG_NameInit.strName[4,7]	:=	'D08Q1'	;
gUI.DiG_NameInit.strName[4,8]	:=	'D08Q2'	;
gUI.DiG_NameInit.strName[5,1]	:=	'D09Q1'	;
gUI.DiG_NameInit.strName[5,2]	:=	'D09Q2'	;
gUI.DiG_NameInit.strName[5,3]	:=	'D10Q1'	;
gUI.DiG_NameInit.strName[5,4]	:=	'D10Q2'	;
gUI.DiG_NameInit.strName[5,5]	:=	'D11Q1'	;
gUI.DiG_NameInit.strName[5,6]	:=	'D11Q2'	;
gUI.DiG_NameInit.strName[5,7]	:=	'D12Q1'	;
gUI.DiG_NameInit.strName[5,8]	:=	'D12Q2'	;
	
gUI.DiG_NameInit.strName[6,1]	:=	'D13Q'	;
gUI.DiG_NameInit.strName[6,2]	:=	'D14Q'	;
gUI.DiG_NameInit.strName[6,3]	:=	'D15Q'	;
gUI.DiG_NameInit.strName[6,4]	:=	'D13L'	;
gUI.DiG_NameInit.strName[6,5]	:=	'D14L'	;
gUI.DiG_NameInit.strName[6,6]	:=	'D15L'	;
gUI.DiG_NameInit.strName[6,7]	:=	'D16L1'	;
gUI.DiG_NameInit.strName[6,8]	:=	'D16L2'	;
	
gUI.DiG_NameInit.strName[7,1]	:=	'D18L'	;
gUI.DiG_NameInit.strName[7,2]	:=	'D19L'	;
gUI.DiG_NameInit.strName[7,3]	:=	'D20L'	;
gUI.DiG_NameInit.strName[7,4]	:=	'D21L'	;
gUI.DiG_NameInit.strName[7,5]	:=	'D22L'	;
gUI.DiG_NameInit.strName[7,6]	:=	'D23L'	;
gUI.DiG_NameInit.strName[7,7]	:=	'D24L'	;
gUI.DiG_NameInit.strName[7,8]	:=	'D25L'	;
gUI.DiG_NameInit.strName[7,9]	:=	'D26L'	;
gUI.DiG_NameInit.strName[7,10]	:=	'D17Q'	;
gUI.DiG_NameInit.strName[7,11]	:=	'D18Q'	;
gUI.DiG_NameInit.strName[7,12]	:=	'D19Q'	;
gUI.DiG_NameInit.strName[7,13]	:=	'D20Q'	;
gUI.DiG_NameInit.strName[7,14]	:=	'D21Q'	;
gUI.DiG_NameInit.strName[7,15]	:=	'D22Q'	;
gUI.DiG_NameInit.strName[7,16]	:=	'D23Q'	;
gUI.DiG_NameInit.strName[7,17]	:=	'D24Q'	;
gUI.DiG_NameInit.strName[7,18]	:=	'D25Q'	;
gUI.DiG_NameInit.strName[7,19]	:=	'D26Q'	;
gUI.DiG_NameInit.strName[7,20]	:=	'D17L1'	;
gUI.DiG_NameInit.strName[7,21]	:=	'D17L2'	;
gUI.DiG_NameInit.strName[7,22]	:=	'D27L1'	;
gUI.DiG_NameInit.strName[7,23]	:=	'D27L2'	;

FOR iVD:=1 TO 7 DO
	FOR iVD1:=1 TO aOil[iVD] DO
		gUI.DiG.arrPV[iVD].sNum[iVD1].strName:=gUI.DiG_NameInit.strName[iVD,iVD1];

	END_FOR
END_FOR
END_ACTION

ACTION initRange:
//标定
(*
gImple.DiG_InitPacket.rExtend[1,1]:=	;
gImple.DiG_InitPacket.rExtend[1,2]:=	;
gImple.DiG_InitPacket.rExtend[1,12]:=	;

gImple.DiG_InitPacket.rRetract[2,1]:=	;
gImple.DiG_InitPacket.rRetract[2,2]:=	;
gImple.DiG_InitPacket.rRetract[2,8]:=	;
*)

FOR iVD:=1 TO 7 DO				//每个比例阀
	FOR iVD1:=1 TO aOil[iVD] DO	//比例阀中每个开关阀
		//-----------------------------------------------
		//gImple.DiG_InitPacket.rRetract[iVD,iVD1]:= 1;//校准数据需重新写入,按照上方注释
		//gImple.DiG_InitPacket.rExtend[iVD,iVD1]:= 200;
		//-----------------------------------------------
		gImple.PV_GroupDi.arrPV[iVD].sNum[iVD1].posVal.Retract:=gImple.DiG_InitPacket.rRetract[iVD,iVD1];
		gImple.PV_GroupDi.arrPV[iVD].sNum[iVD1].posVal.Extend:=gImple.DiG_InitPacket.rExtend[iVD,iVD1];		
		
	END_FOR
END_FOR
(*地轨部分未核对
gImple.DiG_InitPacket.numHead[1,1]:=1;
gImple.DiG_InitPacket.numHead[1,2]:=3;
gImple.DiG_InitPacket.numHead[1,3]:=5;
gImple.DiG_InitPacket.numHead[1,4]:=7;
gImple.DiG_InitPacket.numHead[1,5]:=9;
gImple.DiG_InitPacket.numHead[1,6]:=10;
gImple.DiG_InitPacket.numHead[1,7]:=12;


gImple.DiG_InitPacket.numHead[2,1]:=1;
gImple.DiG_InitPacket.numHead[2,2]:=4;
gImple.DiG_InitPacket.numHead[2,3]:=5;
gImple.DiG_InitPacket.numHead[2,4]:=8;
gImple.DiG_InitPacket.numHead[2,5]:=9;
gImple.DiG_InitPacket.numHead[2,6]:=0;
gImple.DiG_InitPacket.numHead[2,7]:=0;

gImple.DiG_InitPacket.numHead[3,1]:=1;
gImple.DiG_InitPacket.numHead[4,1]:=1;
gImple.DiG_InitPacket.numHead[5,1]:=1;

FOR iVD:=3 TO 5 DO
	FOR iVD1:=2 TO 7 DO
		gImple.DiG_InitPacket.numHead[iVD,iVD1]:=0;
	END_FOR
END_FOR

gImple.DiG_InitPacket.numHead[6,1]:=1;
gImple.DiG_InitPacket.numHead[6,2]:=3;
gImple.DiG_InitPacket.numHead[6,3]:=4;
gImple.DiG_InitPacket.numHead[6,4]:=6;
gImple.DiG_InitPacket.numHead[6,5]:=7;
gImple.DiG_InitPacket.numHead[6,6]:=0;
gImple.DiG_InitPacket.numHead[6,7]:=0;

gImple.DiG_InitPacket.numHead[7,1]:=1;
gImple.DiG_InitPacket.numHead[7,2]:=5;
gImple.DiG_InitPacket.numHead[7,3]:=6;
gImple.DiG_InitPacket.numHead[7,4]:=10;
gImple.DiG_InitPacket.numHead[7,5]:=15;
gImple.DiG_InitPacket.numHead[7,6]:=20;
gImple.DiG_InitPacket.numHead[7,7]:=22;

//----------

gImple.DiG_InitPacket.numTail[1,1]:=2;
gImple.DiG_InitPacket.numTail[1,2]:=4;
gImple.DiG_InitPacket.numTail[1,3]:=5;
gImple.DiG_InitPacket.numTail[1,4]:=7;
gImple.DiG_InitPacket.numTail[1,5]:=8;
gImple.DiG_InitPacket.numTail[1,6]:=9;
gImple.DiG_InitPacket.numTail[1,7]:=0;


gImple.DiG_InitPacket.numTail[2,1]:=3;
gImple.DiG_InitPacket.numTail[2,2]:=4;
gImple.DiG_InitPacket.numTail[2,3]:=7;
gImple.DiG_InitPacket.numTail[2,4]:=8;
gImple.DiG_InitPacket.numTail[2,5]:=11;
gImple.DiG_InitPacket.numTail[2,6]:=0;
gImple.DiG_InitPacket.numTail[2,7]:=0;

gImple.DiG_InitPacket.numTail[3,1]:=8;
gImple.DiG_InitPacket.numTail[4,1]:=8;
gImple.DiG_InitPacket.numTail[5,1]:=8;

FOR iVD:=3 TO 5 DO
	FOR iVD1:=2 TO 7 DO
		gImple.DiG_InitPacket.numTail[iVD,iVD1]:=0;
	END_FOR
END_FOR

gImple.DiG_InitPacket.numTail[6,1]:=2;
gImple.DiG_InitPacket.numTail[6,2]:=3;
gImple.DiG_InitPacket.numTail[6,3]:=5;
gImple.DiG_InitPacket.numTail[6,4]:=6;
gImple.DiG_InitPacket.numTail[6,5]:=8;
gImple.DiG_InitPacket.numTail[6,6]:=0;
gImple.DiG_InitPacket.numTail[6,7]:=0;

gImple.DiG_InitPacket.numTail[7,1]:=4;
gImple.DiG_InitPacket.numTail[7,2]:=5;
gImple.DiG_InitPacket.numTail[7,3]:=9;
gImple.DiG_InitPacket.numTail[7,4]:=14;
gImple.DiG_InitPacket.numTail[7,5]:=19;
gImple.DiG_InitPacket.numTail[7,6]:=21;
gImple.DiG_InitPacket.numTail[7,7]:=23;

FOR iVD:=1 TO 7 DO				//每个比例阀
	FOR iVD1:=1 TO aNo[iVD] DO	//比例阀中每个开关阀
		IF gImple.DiG_InitPacket.numHead[iVD,iVD1]>0 THEN
			
			gImple.DiG_InitPacket.numInColumn[iVD,iVD1]:= gImple.DiG_InitPacket.numTail[iVD,iVD1]-gImple.DiG_InitPacket.numHead[iVD,iVD1]+1;
			
		END_IF
	END_FOR	
END_FOR
*)
END_ACTION

METHOD statusPercentCalcDi : REAL
VAR_INPUT
	psDiG				:POINTER TO propValveModule_Di;	
	iDTDNum				:INT;
	iIndex				:INT;		//比例阀中的索引值（从1开始）
END_VAR
VAR
	rTotal				:REAL;
	rGone				:REAL;
END_VAR

rGone:=psDiG^.arrPV[iDTDNum].sNum[iIndex].posVal.Current-psDiG^.arrPV[iDTDNum].sNum[iIndex].posVal.Retract;
rTotal:=psDiG^.arrPV[iDTDNum].sNum[iIndex].posVal.Extend-psDiG^.arrPV[iDTDNum].sNum[iIndex].posVal.Retract;

statusPercentCalcDi:=rGone/rTotal;
END_METHOD

END_PROGRAM

// Device/Application/can/swmc_floor_rail/swmc_C00_Rx
FUNCTION swmc_C00_Rx : BOOL
VAR_INPUT
	CNT				: UINT;
	psYyz			: POINTER TO YyStation;
END_VAR
VAR
	frame	    : Can_baseframe;
	COB_ID		: UINT;
	I			: UINT;
	Pre			: UINT;
END_VAR

IF gCan.C0RxMsg.RxCounter <>  gCan.C0RxCounter THEN    //接收到新的数据
	
	FOR  I :=1 TO  gCan.C0RxMsg.NoOfRxMessages DO
		frame :=CAN_Read_Data_SWMC(0,I);
		COB_ID :=	frame.id;    //获取ID
		CASE  COB_ID OF     //根据ID解析协议
			//C0-0x300
			16#300:           //液压站状态数据
				psYyz^.Status.HydraulicStation_Power := frame.data[1].0;     //液压站上电 
				psYyz^.Status.Control_Power :=frame.data[1].1;				 //控制总电源上电
				psYyz^.Status.OilPumpM_Fault :=frame.data[2].0;			 //油泵电机故障
				psYyz^.Status.InverterFan_Run :=frame.data[2].1;			 //变频风机
				psYyz^.Status.InverterFan_Fault :=frame.data[3].0;			 //变频风机故障
				psYyz^.Status.OilPumpFan :=frame.data[3].1;					 //SP油泵风机故障
				psYyz^.Status.FrequencyConversion_Fault :=frame.data[4].0;   //变频故障
				psYyz^.Status.FrequencyConversion_Run :=frame.data[4].1;	 //变频运行
				
			//C0-0x301
			16#301:           //液压站状态数据
				Pre :=BYTE_TO_WORD(frame.data[1]) OR SHL(BYTE_TO_WORD(frame.data[2]),8);
	 			psYyz^.Status.pressureStatus:= 	(Pre-4000)/16000.0*400;	
				Pre :=BYTE_TO_WORD(frame.data[3]) OR SHL(BYTE_TO_WORD(frame.data[4]),8);
				
			 	//???
				psYyz^.Status.yeweiStatus				:=frame.data[5].0;
				(*
				psYyz^.Status.FrequencyConversion_Fault	:=frame.data[7].0;
				psYyz^.Status.FrequencyConversion_Run	:=frame.data[7].1;
				psYyz^.Status.HydraulicStation_Power	:=frame.data[7].2;
				psYyz^.Status.Control_Power				:=frame.data[7].3;
				psYyz^.Status.InverterFan_Run			:=frame.data[7].4;
				psYyz^.Status.OilPumpFan				:=frame.data[7].5;
				psYyz^.Status.OilPumpMotor_Fault		:=frame.data[7].6;
				psYyz^.Status.InverterFan_Fault			:=frame.data[7].7;
				*)	
		END_CASE
	END_FOR
	gCan.C0RxCounter := gCan.C0RxMsg.RxCounter ;
END_IF

END_FUNCTION

// Device/Application/can/swmc_floor_rail/swmc_C00_Tx
FUNCTION swmc_C00_Tx : BOOL
VAR_INPUT
	CNT				: UINT;
	psYyz			: POINTER TO YyStation;
END_VAR
VAR
	senddata	: ARRAY[1..8] OF BYTE;
	Send_cnt	: UINT;
END_VAR

//控制速度--待定
Send_cnt :=  CNT MOD 3;

CASE Send_cnt OF
	
    1:
	 //C0-0x400
	 
	senddata[1].0 :=  psYyz^.Cmd.InverterFan_Ctrl; 		// 变频风机控制
	senddata[1].1 :=  psYyz^.Cmd.OilPumpFan_Ctrl;		// 油泵风机控制
	senddata[2].0 :=  psYyz^.Cmd.OilPumpMotor_Ctrl;		// 油泵电机控制    
	senddata[2].1 :=  psYyz^.Cmd.OilPumpMotor_PN_Ctrl;  // 油泵电机正反转
	senddata[3].0 :=  psYyz^.Cmd.HL_Mode_Ctrl;          // 高低速模式
	senddata[3].1 :=  psYyz^.Cmd.KEEP_Mode_Ctrl;        // 恒速模式      
	senddata[4].0 :=  0;                     			//储能开关
	senddata[5]   :=  WORD_TO_BYTE(psYyz^.Cmd.Oil_Pre_Val);      		           
	senddata[6]   :=  WORD_TO_BYTE(SHR(psYyz^.Cmd.Oil_Pre_Val,8));    //油压控制   
	senddata[7]   :=  0;           //设置A04存储夹紧块状态
	senddata[8]   :=  0; 

	 (*
	senddata[1].0 :=  psYyz^.Cmd.InverterFan_Ctrl; 		// 变频风机控制
	senddata[1].1 :=  psYyz^.Cmd.OilPumpFan_Ctrl;		// 油泵风机控制
	senddata[2]   :=  0;  
	senddata[3]   :=  0;    
	senddata[4]	  :=  0;                     			
	senddata[5]   :=  0;      		           
	senddata[6]   :=  0; 
	senddata[7]   :=  0;           
	senddata[8]   :=  0; 
	*)
	
	//发送至C0
	CAN_Send_Data_SWMC(0, 16#400,senddata);   //发送ID 0x400到 C0

END_CASE

END_FUNCTION

// Device/Application/can/swmc_floor_rail/swmc_C01_Rx
FUNCTION swmc_C01_Rx : BOOL
VAR_INPUT
	CNT				: UINT;
	psYyz			: POINTER TO YyStation;
	psPVDi			: POINTER TO propValveModule_Di;
	
	
END_VAR
VAR
	frame	 	    : Can_baseframe;
	COB_ID			: UINT;
	I				: UINT;
	pos				: WORD;
	Pre				: UINT;
END_VAR

IF gCan.C1RxMsg.RxCounter <>  gCan.C1RxCounter THEN    //接收到新的数据

	FOR  I := 1 TO  gCan.C1RxMsg.NoOfRxMessages DO
		frame :=CAN_Read_Data_SWMC(1,I);
		COB_ID :=	frame.id;    //获取ID
		CASE COB_ID OF     //根据ID解析协议
		
			
			//C1-0x310
			16#310:           //接收C1送来的数据
				pos := BYTE_TO_WORD(frame.data[1]) OR SHL(BYTE_TO_WORD(frame.data[2]),8);  	
				//psDiG3^.RVD3[1].status.posVal.Current
				psPVDi^.arrPV[3].sNum[1].posVal.Current:= pos*0.1;
				//psDiG3^.RVD3[1].status.posVal.Current:= pos*0.1;	//驱动插销油缸D01Q1-位移传感器	
				pos := BYTE_TO_WORD(frame.data[3]) OR SHL(BYTE_TO_WORD(frame.data[4]),8);  	
				psPVDi^.arrPV[3].sNum[2].posVal.Current:= pos*0.1;	//驱动插销油缸D01Q2-位移传感器	
				pos := BYTE_TO_WORD(frame.data[5]) OR SHL(BYTE_TO_WORD(frame.data[6]),8);  	
				psPVDi^.arrPV[3].sNum[3].posVal.Current:= pos*0.1;	//驱动插销油缸D02Q1-位移传感器	
				pos := BYTE_TO_WORD(frame.data[7]) OR SHL(BYTE_TO_WORD(frame.data[8]),8);  	
				psPVDi^.arrPV[3].sNum[4].posVal.Current:= pos*0.1;	//驱动插销油缸D02Q2-位移传感器	
			//C1-0x311
			16#311:           //接收C1送来的数据
				pos := BYTE_TO_WORD(frame.data[1]) OR SHL(BYTE_TO_WORD(frame.data[2]),8);  	
				psPVDi^.arrPV[3].sNum[5].posVal.Current:= pos*0.1;	//驱动插销油缸D03Q1-位移传感器	
				pos := BYTE_TO_WORD(frame.data[3]) OR SHL(BYTE_TO_WORD(frame.data[4]),8);  	
				psPVDi^.arrPV[3].sNum[6].posVal.Current:= pos*0.1;	//驱动插销油缸D03Q2-位移传感器	
				pos := BYTE_TO_WORD(frame.data[5]) OR SHL(BYTE_TO_WORD(frame.data[6]),8);  	
				psPVDi^.arrPV[3].sNum[7].posVal.Current:= pos*0.1;	//驱动插销油缸D04Q1-位移传感器	
				pos := BYTE_TO_WORD(frame.data[7]) OR SHL(BYTE_TO_WORD(frame.data[8]),8);  	
				psPVDi^.arrPV[3].sNum[8].posVal.Current:= pos*0.1;	//驱动插销油缸D04Q2-位移传感器
				
		//比例阀DTD4	
			//C1-0x312
			16#312:           //接收C1送来的数据
				pos := BYTE_TO_WORD(frame.data[1]) OR SHL(BYTE_TO_WORD(frame.data[2]),8);  	
				psPVDi^.arrPV[4].sNum[1].posVal.Current:= pos*0.1;	//驱动插销油缸D05Q1-位移传感器	
				pos := BYTE_TO_WORD(frame.data[3]) OR SHL(BYTE_TO_WORD(frame.data[4]),8);  	
				psPVDi^.arrPV[4].sNum[2].posVal.Current:= pos*0.1;	//驱动插销油缸D05Q2-位移传感器	
				pos := BYTE_TO_WORD(frame.data[5]) OR SHL(BYTE_TO_WORD(frame.data[6]),8);  	
				psPVDi^.arrPV[4].sNum[3].posVal.Current:= pos*0.1;	//驱动插销油缸D06Q1-位移传感器	
				pos := BYTE_TO_WORD(frame.data[7]) OR SHL(BYTE_TO_WORD(frame.data[8]),8);  	
				psPVDi^.arrPV[4].sNum[4].posVal.Current:= pos*0.1;	//驱动插销油缸D06Q2-位移传感器	
			//C1-0x313
			16#313:           //接收C1送来的数据
				pos := BYTE_TO_WORD(frame.data[1]) OR SHL(BYTE_TO_WORD(frame.data[2]),8);  	
				psPVDi^.arrPV[4].sNum[5].posVal.Current:= pos*0.1;	//驱动插销油缸D07Q1-位移传感器	
				pos := BYTE_TO_WORD(frame.data[3]) OR SHL(BYTE_TO_WORD(frame.data[4]),8);  	
				psPVDi^.arrPV[4].sNum[6].posVal.Current:= pos*0.1;	//驱动插销油缸D07Q2-位移传感器	
				pos := BYTE_TO_WORD(frame.data[5]) OR SHL(BYTE_TO_WORD(frame.data[6]),8);  	
				psPVDi^.arrPV[4].sNum[7].posVal.Current:= pos*0.1;	//驱动插销油缸D08Q1-位移传感器	
				pos := BYTE_TO_WORD(frame.data[7]) OR SHL(BYTE_TO_WORD(frame.data[8]),8);  	
				psPVDi^.arrPV[4].sNum[8].posVal.Current:= pos*0.1;	//驱动插销油缸D08Q2-位移传感器
				
		//比例阀DTD5					
			//C1-0x314
			16#314:           //接收C1送来的数据
				pos := BYTE_TO_WORD(frame.data[1]) OR SHL(BYTE_TO_WORD(frame.data[2]),8);  	
				psPVDi^.arrPV[5].sNum[1].posVal.Current:= pos*0.1;	//驱动插销油缸D09Q1-位移传感器	
				pos := BYTE_TO_WORD(frame.data[3]) OR SHL(BYTE_TO_WORD(frame.data[4]),8);  	
				psPVDi^.arrPV[5].sNum[2].posVal.Current:= pos*0.1;	//驱动插销油缸D09Q2-位移传感器	
				pos := BYTE_TO_WORD(frame.data[5]) OR SHL(BYTE_TO_WORD(frame.data[6]),8);  	
				psPVDi^.arrPV[5].sNum[3].posVal.Current:= pos*0.1;	//驱动插销油缸D10Q1-位移传感器	
				pos := BYTE_TO_WORD(frame.data[7]) OR SHL(BYTE_TO_WORD(frame.data[8]),8);  	
				psPVDi^.arrPV[5].sNum[4].posVal.Current:= pos*0.1;	//驱动插销油缸D10Q2-位移传感器	
			//C1-0x315
			16#315:           //接收C1送来的数据
				pos := BYTE_TO_WORD(frame.data[1]) OR SHL(BYTE_TO_WORD(frame.data[2]),8);  	
				psPVDi^.arrPV[5].sNum[5].posVal.Current:= pos*0.1;	//驱动插销油缸D11Q1-位移传感器	
				pos := BYTE_TO_WORD(frame.data[3]) OR SHL(BYTE_TO_WORD(frame.data[4]),8);  	
				psPVDi^.arrPV[5].sNum[6].posVal.Current:= pos*0.1;	//驱动插销油缸D11Q2-位移传感器	
				pos := BYTE_TO_WORD(frame.data[5]) OR SHL(BYTE_TO_WORD(frame.data[6]),8);  	
				psPVDi^.arrPV[5].sNum[7].posVal.Current:= pos*0.1;	//驱动插销油缸D12Q1-位移传感器	
				pos := BYTE_TO_WORD(frame.data[7]) OR SHL(BYTE_TO_WORD(frame.data[8]),8);  	
				psPVDi^.arrPV[5].sNum[8].posVal.Current:= pos*0.1;	//驱动插销油缸D12Q2-位移传感器
			
			//C1-0x316
			16#316:           //液压站状态数据
			
				Pre :=BYTE_TO_WORD(frame.data[1]) OR SHL(BYTE_TO_WORD(frame.data[2]),8);
	 			psYyz^.Status.pressureV2:= 	(Pre-4000)/16000.0*400;	
				
			    Pre :=BYTE_TO_WORD(frame.data[3]) OR SHL(BYTE_TO_WORD(frame.data[4]),8);
	 			psYyz^.Status.pressureV3:= 	(Pre-4000)/16000.0*400;	
				
			
			
			(*
				Pre :=BYTE_TO_WORD(frame.data[1]) OR SHL(BYTE_TO_WORD(frame.data[2]),8);
	 			psYyz^.Status.pressureStatus:= 	(Pre-4000)/16000.0*400;	
				Pre :=BYTE_TO_WORD(frame.data[3]) OR SHL(BYTE_TO_WORD(frame.data[4]),8);
			 	//???
				psYyz^.Status.yeweiStatus				:=frame.data[5].0;
				
				psYyz^.Status.FrequencyConversion_Fault	:=frame.data[7].0;
				psYyz^.Status.FrequencyConversion_Run	:=frame.data[7].1;
				psYyz^.Status.HydraulicStation_Power	:=frame.data[7].2;
				psYyz^.Status.Control_Power				:=frame.data[7].3;
				psYyz^.Status.InverterFan_Run			:=frame.data[7].4;
				psYyz^.Status.OilPumpFan				:=frame.data[7].5;
				psYyz^.Status.OilPumpMotor_Fault		:=frame.data[7].6;
				psYyz^.Status.InverterFan_Fault			:=frame.data[7].7;
					*)	
		END_CASE
	END_FOR


	gCan.C0RxCounter := gCan.C0RxMsg.RxCounter ;
END_IF

END_FUNCTION

// Device/Application/can/swmc_floor_rail/swmc_C01_Tx
FUNCTION swmc_C01_Tx : BOOL
VAR_INPUT
	CNT				: UINT;
	psPVDi			: POINTER TO propValveModule_Di;
	
END_VAR
VAR
	senddata	: ARRAY[1..8] OF BYTE;
	Send_cnt	: UINT;
END_VAR

//控制速度--待定
Send_cnt :=  CNT MOD 3;

CASE Send_cnt OF
	
    1:
	 //C1-0x410
	 
	senddata[1] :=  WORD_TO_BYTE(psPVDi^.arrPV[1].percenVal);  		   //发送DTD1比例阀值
	senddata[2] :=  WORD_TO_BYTE(SHR(psPVDi^.arrPV[1].percenVal,8));    //0-65535  对应0-100  
	senddata[3] :=  WORD_TO_BYTE(psPVDi^.arrPV[2].percenVal);  		   //发送DTD2比例阀值
	senddata[4] :=  WORD_TO_BYTE(SHR(psPVDi^.arrPV[2].percenVal,8));    //0-65535  对应0-100  
	senddata[5] :=  WORD_TO_BYTE(psPVDi^.arrPV[3].percenVal);  		   //发送DTD3比例阀值
	senddata[6] :=  WORD_TO_BYTE(SHR(psPVDi^.arrPV[3].percenVal,8));    //0-65535  对应0-100  
	senddata[7] :=  WORD_TO_BYTE(psPVDi^.arrPV[4].percenVal);  		   //发送DTD4比例阀值
	senddata[8] :=  WORD_TO_BYTE(SHR(psPVDi^.arrPV[4].percenVal,8));    //0-65535  对应0-100  
	//发送至C1
	CAN_Send_Data_SWMC(1, 16#410,senddata);   //发送ID 0x410到C1
	
	2:
	 //C1-0x411
	senddata[1] :=  WORD_TO_BYTE(psPVDi^.arrPV[5].percenVal);  		   //发送DTD5比例阀值
	senddata[2] :=  WORD_TO_BYTE(SHR(psPVDi^.arrPV[5].percenVal,8));    //0-65535  对应0-100  
	
	senddata[3].0:=  psPVDi^.arrPV[1].sColumn[1].bE_Open;               
	senddata[3].1:=  psPVDi^.arrPV[1].sColumn[1].bR_Open;			//send D00Q1&D00Q2
	senddata[3].2:=  psPVDi^.arrPV[1].sColumn[2].bE_Open;               
	senddata[3].3:=  psPVDi^.arrPV[1].sColumn[2].bR_Open;			//send D28L1&D28L2
	
	senddata[4].0:=  psPVDi^.arrPV[1].sColumn[3].bE_Open;               
	senddata[4].1:=  psPVDi^.arrPV[1].sColumn[3].bR_Open;			//send D29L&D30L
	senddata[4].2:=  psPVDi^.arrPV[1].sColumn[4].bE_Open;               
	senddata[4].3:=  psPVDi^.arrPV[1].sColumn[4].bR_Open;			//send D00L1&00L2
	
	senddata[5].0:=  psPVDi^.arrPV[1].sColumn[5].bE_Open;               
	senddata[5].1:=  psPVDi^.arrPV[1].sColumn[5].bR_Open;           //send D01L
	senddata[5].2:=  psPVDi^.arrPV[1].sColumn[6].bE_Open;               
	senddata[5].3:=  psPVDi^.arrPV[1].sColumn[6].bR_Open;           //send D28Q&29Q
	
	senddata[6].0:=  psPVDi^.arrPV[1].sColumn[7].bE_Open;               
	senddata[6].1:=  psPVDi^.arrPV[1].sColumn[7].bR_Open;           //send D30Q
	//发送至C1
	CAN_Send_Data_SWMC(1, 16#411,senddata);				//发送ID 0x411到C1
	
	3:
	 //C1.1 IO-0x412
	senddata[1].0:=  psPVDi^.arrPV[2].sColumn[1].bE_Open;               
	senddata[1].1:=  psPVDi^.arrPV[2].sColumn[1].bR_Open;           //send D02L&D03L||D04L
	
	senddata[2].0:=  psPVDi^.arrPV[3].sColumn[1].bE_Open;               
	senddata[2].1:=  psPVDi^.arrPV[3].sColumn[1].bR_Open; 	        //send D01Q1&D01Q2||02~04QX

	senddata[3].0:=  psPVDi^.arrPV[4].sColumn[1].bE_Open;               
	senddata[3].1:=  psPVDi^.arrPV[4].sColumn[1].bR_Open;			//send D05Q1&05Q2||06~08QX
		
	senddata[4].0:=  psPVDi^.arrPV[5].sColumn[1].bE_Open;               
	senddata[4].1:=  psPVDi^.arrPV[5].sColumn[1].bR_Open;			//send D09Q1&09Q2||10~12QX
	//发送至C1
	CAN_Send_Data_SWMC(1, 16#412,senddata);				//发送ID 0x412到C1.1
	
	4:
	 //C1.2 IO-0x413
	senddata[1].0:=  psPVDi^.arrPV[2].sColumn[2].bE_Open;               
	senddata[1].1:=  psPVDi^.arrPV[2].sColumn[2].bR_Open;           //send D05L
	
	senddata[2].0:=  psPVDi^.arrPV[2].sColumn[3].bE_Open;               
	senddata[2].1:=  psPVDi^.arrPV[2].sColumn[3].bR_Open; 	        //send D06L&D07L||D08L

	senddata[3].0:=  psPVDi^.arrPV[2].sColumn[4].bE_Open;               
	senddata[3].1:=  psPVDi^.arrPV[2].sColumn[4].bR_Open;			//send D09L
		
	senddata[4].0:=  psPVDi^.arrPV[2].sColumn[5].bE_Open;               
	senddata[4].1:=  psPVDi^.arrPV[2].sColumn[5].bR_Open;			//send D010L&11L||D12L
	//发送至C1
	CAN_Send_Data_SWMC(1, 16#413,senddata);				//发送ID 0x413到C1.2

END_CASE

END_FUNCTION

// Device/Application/can/swmc_floor_rail/swmc_C02_Rx
FUNCTION swmc_C02_Rx : BOOL
VAR_INPUT
	CNT				: UINT;
	psYyz			: POINTER TO YyStation;
	psPVDi			: POINTER TO propValveModule_Di;
END_VAR
VAR
	frame	 	    : Can_baseframe;
	COB_ID			: UINT;
	I				: UINT;
	pos				: WORD;
END_VAR

IF gCan.C2RxMsg.RxCounter <>  gCan.C2RxCounter THEN    //接收到新的数据

	FOR  I := 1 TO  gCan.C2RxMsg.NoOfRxMessages DO
		frame :=CAN_Read_Data_SWMC(2,I);
		COB_ID :=	frame.id;    //获取ID
		CASE COB_ID OF     //根据ID解析协议
	
			//C1-0x320
			16#320:           //接收C2送来的数据
				pos := BYTE_TO_WORD(frame.data[1]) OR SHL(BYTE_TO_WORD(frame.data[2]),8);  	
				psPVDi^.arrPV[7].sNum[1].posVal.Current:= pos*0.1;	//驱动插销油缸D18L-位移传感器	
				pos := BYTE_TO_WORD(frame.data[3]) OR SHL(BYTE_TO_WORD(frame.data[4]),8);  	
				psPVDi^.arrPV[7].sNum[2].posVal.Current:= pos*0.1;	//驱动插销油缸D19L-位移传感器	
				pos := BYTE_TO_WORD(frame.data[5]) OR SHL(BYTE_TO_WORD(frame.data[6]),8);  	
				psPVDi^.arrPV[7].sNum[3].posVal.Current:= pos*0.1;	//驱动插销油缸D20L-位移传感器		
				pos := BYTE_TO_WORD(frame.data[7]) OR SHL(BYTE_TO_WORD(frame.data[8]),8);  	
				psPVDi^.arrPV[7].sNum[4].posVal.Current:= pos*0.1;	//驱动插销油缸D21L-位移传感器		
			//C1-0x321
			16#321:           //接收C2送来的数据
				pos := BYTE_TO_WORD(frame.data[1]) OR SHL(BYTE_TO_WORD(frame.data[2]),8);  	
				psPVDi^.arrPV[7].sNum[5].posVal.Current:= pos*0.1;	//驱动插销油缸D22L-位移传感器	
				pos := BYTE_TO_WORD(frame.data[3]) OR SHL(BYTE_TO_WORD(frame.data[4]),8);  	
				psPVDi^.arrPV[7].sNum[6].posVal.Current:= pos*0.1;	//驱动插销油缸D23L-位移传感器	
				pos := BYTE_TO_WORD(frame.data[5]) OR SHL(BYTE_TO_WORD(frame.data[6]),8);  	
				psPVDi^.arrPV[7].sNum[7].posVal.Current:= pos*0.1;	//驱动插销油缸D24L-位移传感器	
				pos := BYTE_TO_WORD(frame.data[7]) OR SHL(BYTE_TO_WORD(frame.data[8]),8);  	
				psPVDi^.arrPV[7].sNum[8].posVal.Current:= pos*0.1;	//驱动插销油缸D25L-位移传感器
			//C1-0x322
			16#322:           //接收C2送来的数据
				pos := BYTE_TO_WORD(frame.data[1]) OR SHL(BYTE_TO_WORD(frame.data[2]),8);  	
				psPVDi^.arrPV[7].sNum[9].posVal.Current:= pos*0.1;	//驱动插销油缸D26L-位移传感器	
				pos := BYTE_TO_WORD(frame.data[3]) OR SHL(BYTE_TO_WORD(frame.data[4]),8);  	
				psPVDi^.arrPV[7].sNum[10].posVal.Current:= pos*0.1;	//驱动插销油缸D17Q-位移传感器	
				pos := BYTE_TO_WORD(frame.data[5]) OR SHL(BYTE_TO_WORD(frame.data[6]),8);  	
				psPVDi^.arrPV[7].sNum[11].posVal.Current:= pos*0.1;	//驱动插销油缸D18Q-位移传感器	
				pos := BYTE_TO_WORD(frame.data[7]) OR SHL(BYTE_TO_WORD(frame.data[8]),8);  	
				psPVDi^.arrPV[7].sNum[12].posVal.Current:= pos*0.1;	//驱动插销油缸D19Q-位移传感器
			16#323:           //接收C2送来的数据
				pos := BYTE_TO_WORD(frame.data[1]) OR SHL(BYTE_TO_WORD(frame.data[2]),8);  	
				psPVDi^.arrPV[7].sNum[13].posVal.Current:= pos*0.1;	//驱动插销油缸D20Q-位移传感器	
				pos := BYTE_TO_WORD(frame.data[3]) OR SHL(BYTE_TO_WORD(frame.data[4]),8);  	
				psPVDi^.arrPV[7].sNum[14].posVal.Current:= pos*0.1;	//驱动插销油缸D21Q-位移传感器	
				pos := BYTE_TO_WORD(frame.data[5]) OR SHL(BYTE_TO_WORD(frame.data[6]),8);  	
				psPVDi^.arrPV[7].sNum[15].posVal.Current:= pos*0.1;	//驱动插销油缸D22Q-位移传感器	
				pos := BYTE_TO_WORD(frame.data[7]) OR SHL(BYTE_TO_WORD(frame.data[8]),8);  	
				psPVDi^.arrPV[7].sNum[16].posVal.Current:= pos*0.1;	//驱动插销油缸D23Q-位移传感器
		
			16#324:           //接收C2送来的数据
				pos := BYTE_TO_WORD(frame.data[1]) OR SHL(BYTE_TO_WORD(frame.data[2]),8);  	
				psPVDi^.arrPV[7].sNum[17].posVal.Current:= pos*0.1;	//驱动插销油缸D24Q-位移传感器	
				pos := BYTE_TO_WORD(frame.data[3]) OR SHL(BYTE_TO_WORD(frame.data[4]),8);  	
				psPVDi^.arrPV[7].sNum[18].posVal.Current:= pos*0.1;	//驱动插销油缸D25Q-位移传感器	
				pos := BYTE_TO_WORD(frame.data[5]) OR SHL(BYTE_TO_WORD(frame.data[6]),8);  	
				psPVDi^.arrPV[7].sNum[19].posVal.Current:= pos*0.1;	//驱动插销油缸D26Q-位移传感器	
				pos := BYTE_TO_WORD(frame.data[7]) OR SHL(BYTE_TO_WORD(frame.data[8]),8);  	
				psPVDi^.arrPV[7].sNum[20].posVal.Current:= pos*0.1;	//驱动插销油缸D17L1-位移传感器
			
			16#325:           //接收C2送来的数据
				pos := BYTE_TO_WORD(frame.data[1]) OR SHL(BYTE_TO_WORD(frame.data[2]),8);  	
				psPVDi^.arrPV[7].sNum[21].posVal.Current:= pos*0.1;	//驱动插销油缸D17L2-位移传感器	
				pos := BYTE_TO_WORD(frame.data[3]) OR SHL(BYTE_TO_WORD(frame.data[4]),8);  	
				psPVDi^.arrPV[7].sNum[22].posVal.Current:= pos*0.1;	//驱动插销油缸D27L1-位移传感器	
				pos := BYTE_TO_WORD(frame.data[5]) OR SHL(BYTE_TO_WORD(frame.data[6]),8);  	
				psPVDi^.arrPV[7].sNum[23].posVal.Current:= pos*0.1;	//驱动插销油缸D27L2-位移传感器

		END_CASE
	END_FOR


	gCan.C2RxCounter := gCan.C2RxMsg.RxCounter ;
END_IF

END_FUNCTION

// Device/Application/can/swmc_floor_rail/swmc_C02_Tx
FUNCTION swmc_C02_Tx : BOOL
VAR_INPUT
	CNT				: UINT;
	psPVDi			: POINTER TO propValveModule_Di;

END_VAR
VAR
	senddata	: ARRAY[1..8] OF BYTE;
	Send_cnt	: UINT;
END_VAR

//速度控制--待定
Send_cnt :=  CNT MOD 3;

CASE Send_cnt OF
	
	1:
 	//C2-0x420
	senddata[1] :=  WORD_TO_BYTE(psPVDi^.arrPV[6].percenVal);  		   //发送DTD6比例阀值
	senddata[2] :=  WORD_TO_BYTE(SHR(psPVDi^.arrPV[6].percenVal,8));    //0-65535  对应0-100  

	senddata[3] :=  WORD_TO_BYTE(psPVDi^.arrPV[7].percenVal);  		   //发送DTD7比例阀值
	senddata[4] :=  WORD_TO_BYTE(SHR(psPVDi^.arrPV[7].percenVal,8));    //0-65535  对应0-100  
	
	senddata[5].0:=  psPVDi^.arrPV[6].sColumn[1].bE_Open;
	senddata[5].1:=  psPVDi^.arrPV[6].sColumn[1].bR_Open;			//send D13Q&14Q
	senddata[5].2:=  psPVDi^.arrPV[6].sColumn[2].bE_Open;
	senddata[5].3:=  psPVDi^.arrPV[6].sColumn[2].bR_Open;			//send D15Q
	
	senddata[6].0:=  psPVDi^.arrPV[6].sColumn[3].bE_Open;
	senddata[6].1:=  psPVDi^.arrPV[6].sColumn[3].bR_Open;			//send D13L&14L
	senddata[6].2:=  psPVDi^.arrPV[6].sColumn[4].bE_Open;
	senddata[6].3:=  psPVDi^.arrPV[6].sColumn[4].bR_Open;			//send D15L
	
	senddata[7].0:=  psPVDi^.arrPV[6].sColumn[5].bE_Open;
	senddata[7].1:=  psPVDi^.arrPV[6].sColumn[5].bR_Open;			//send D16L1&16L2
	senddata[7].2:=  psPVDi^.arrPV[7].sColumn[1].bE_Open;
	senddata[7].3:=  psPVDi^.arrPV[7].sColumn[1].bR_Open;			//send D18L&19L||L20~21L
	
	senddata[8].0:=  psPVDi^.arrPV[7].sColumn[2].bE_Open;
	senddata[8].1:=  psPVDi^.arrPV[7].sColumn[2].bR_Open;			//send D22L1&22L2
	senddata[8].2:=  psPVDi^.arrPV[7].sColumn[3].bE_Open;
	senddata[8].3:=  psPVDi^.arrPV[7].sColumn[3].bR_Open;			//send D23L&24L||25L~26L
	
	
	//发送至C2
	CAN_Send_Data_SWMC(2, 16#420,senddata);				//发送ID 0x420到C2
	
	2:
 	//C2-0x421
		
	//senddata[1].0:=  psDiG7^.D18Q.cmd.E_Open;
	//senddata[1].1:=  psDiG7^.D19Q.cmd.R_Open;			//send D18Q&19Q||20Q~21Q
	senddata[1].0:=  psPVDi^.arrPV[7].sColumn[4].bE_Open;
	senddata[1].1:=  psPVDi^.arrPV[7].sColumn[4].bR_Open;			//send D18Q&19Q||20Q~21Q
		
	senddata[2].0:=  psPVDi^.arrPV[7].sColumn[5].bE_Open;
	senddata[2].1:=  psPVDi^.arrPV[7].sColumn[5].bR_Open;			//send D22Q&23Q||24Q~26Q
	
	senddata[3].0:=  psPVDi^.arrPV[7].sColumn[6].bE_Open;
	senddata[3].1:=  psPVDi^.arrPV[7].sColumn[6].bR_Open;			//send D17L1&17L2
	
	senddata[4].0:=  psPVDi^.arrPV[7].sColumn[7].bE_Open;
	senddata[4].1:=  psPVDi^.arrPV[7].sColumn[7].bR_Open;			//send D27L1&27L2
	
	//发送至C2.1-IO
	CAN_Send_Data_SWMC(2, 16#421,senddata);				//发送ID 0x420到C2.1-IO
	
	
END_CASE

END_FUNCTION

// Device/Application/can/swmc_floor_rail/swmc_C09_Rx
FUNCTION swmc_C09_Rx : BOOL
VAR_INPUT
	CNT				: UINT;
	psYyz			: POINTER TO YyStation;
	psPVDi			: POINTER TO propValveModule_Di;
	
END_VAR
VAR
	frame	 	    : Can_baseframe;
	COB_ID			: UINT;
	I				: UINT;
	pos				: WORD;
END_VAR

IF gCan.C9RxMsg.RxCounter <>  gCan.C9RxCounter THEN    //接收到新的数据

	FOR  I := 1 TO  gCan.C9RxMsg.NoOfRxMessages DO
		frame :=CAN_Read_Data_SWMC(9,I);
		COB_ID :=	frame.id;    //获取ID
		CASE COB_ID OF     //根据ID解析协议
		
		//比例阀DTD1
			//C11-0x3B0
			16#3B0:           //接收C9送来的数据
				pos := BYTE_TO_WORD(frame.data[1]) OR SHL(BYTE_TO_WORD(frame.data[2]),8);  	
							//C9-0x390
			16#390:           //接收C9送来的数据
				pos   := BYTE_TO_WORD(frame.data[1]) OR SHL(BYTE_TO_WORD(frame.data[2]),8);  	
				psPVDi^.arrPV[1].sNum[3].posVal.Current  := pos*0.1;	//驱动插销油缸D28L1-位移传感器	
				pos   := BYTE_TO_WORD(frame.data[3]) OR SHL(BYTE_TO_WORD(frame.data[4]),8);  	
				psPVDi^.arrPV[1].sNum[4].posVal.Current  := pos*0.1;	//驱动插销油缸D28L2-位移传感器	
				pos   := BYTE_TO_WORD(frame.data[5]) OR SHL(BYTE_TO_WORD(frame.data[6]),8);  	
				psPVDi^.arrPV[1].sNum[5].posVal.Current  := pos*0.1;	//驱动插销油缸D29L-位移传感器		
				pos   := BYTE_TO_WORD(frame.data[7]) OR SHL(BYTE_TO_WORD(frame.data[8]),8);  	
				psPVDi^.arrPV[1].sNum[6].posVal.Current  := pos*0.1;	//驱动插销油缸D30L-位移传感器		
			
			16#391:           //接收C9送来的数据
				pos   := BYTE_TO_WORD(frame.data[1]) OR SHL(BYTE_TO_WORD(frame.data[2]),8);  	
				psPVDi^.arrPV[1].sNum[9].posVal.Current := pos*0.1;	//驱动插销油缸D01L-位移传感器	
				pos   := BYTE_TO_WORD(frame.data[3]) OR SHL(BYTE_TO_WORD(frame.data[4]),8);  	
				psPVDi^.arrPV[1].sNum[10].posVal.Current := pos*0.1;	//驱动插销油缸D28Q-位移传感器	
				pos   := BYTE_TO_WORD(frame.data[5]) OR SHL(BYTE_TO_WORD(frame.data[6]),8);  	
				psPVDi^.arrPV[1].sNum[11].posVal.Current := pos*0.1;	//驱动插销油缸D29Q-位移传感器		
				pos   := BYTE_TO_WORD(frame.data[7]) OR SHL(BYTE_TO_WORD(frame.data[8]),8);  	
				psPVDi^.arrPV[1].sNum[12].posVal.Current := pos*0.1;	//驱动插销油缸D30Q-位移传感器		
				
			16#392:           //接收C9送来的数据
				pos   := BYTE_TO_WORD(frame.data[1]) OR SHL(BYTE_TO_WORD(frame.data[2]),8);  	
				psPVDi^.arrPV[1].sNum[7].posVal.Current := pos*0.1;	//驱动插销油缸D00L1-位移传感器	
				pos   := BYTE_TO_WORD(frame.data[3]) OR SHL(BYTE_TO_WORD(frame.data[4]),8);  	
				psPVDi^.arrPV[2].sNum[1].posVal.Current  := pos*0.1;	//驱动插销油缸D02L-位移传感器	
				pos   := BYTE_TO_WORD(frame.data[5]) OR SHL(BYTE_TO_WORD(frame.data[6]),8);  	
				psPVDi^.arrPV[2].sNum[2].posVal.Current  := pos*0.1;	//驱动插销油缸D03L-位移传感器		
				pos   := BYTE_TO_WORD(frame.data[7]) OR SHL(BYTE_TO_WORD(frame.data[8]),8);  	
				psPVDi^.arrPV[2].sNum[3].posVal.Current  := pos*0.1;	//驱动插销油缸D04L-位移传感器		
				
			16#393:           //接收C9送来的数据
				pos   := BYTE_TO_WORD(frame.data[1]) OR SHL(BYTE_TO_WORD(frame.data[2]),8);  	
				psPVDi^.arrPV[2].sNum[4].posVal.Current  := pos*0.1;	//驱动插销油缸D05L-位移传感器	
				pos   := BYTE_TO_WORD(frame.data[3]) OR SHL(BYTE_TO_WORD(frame.data[4]),8);  	
				psPVDi^.arrPV[2].sNum[5].posVal.Current  := pos*0.1;	//驱动插销油缸D06L-位移传感器	
				pos   := BYTE_TO_WORD(frame.data[5]) OR SHL(BYTE_TO_WORD(frame.data[6]),8);  	
				psPVDi^.arrPV[2].sNum[6].posVal.Current  := pos*0.1;	//驱动插销油缸D07L-位移传感器		
				pos   := BYTE_TO_WORD(frame.data[7]) OR SHL(BYTE_TO_WORD(frame.data[8]),8);  	
				psPVDi^.arrPV[2].sNum[7].posVal.Current  := pos*0.1;	//驱动插销油缸D08L-位移传感器		

			16#394:           //接收C9送来的数据
				pos   := BYTE_TO_WORD(frame.data[1]) OR SHL(BYTE_TO_WORD(frame.data[2]),8);  	
				psPVDi^.arrPV[2].sNum[8].posVal.Current  := pos*0.1;	//驱动插销油缸D09L-位移传感器	
				pos   := BYTE_TO_WORD(frame.data[3]) OR SHL(BYTE_TO_WORD(frame.data[4]),8);  	
				psPVDi^.arrPV[2].sNum[9].posVal.Current  := pos*0.1;	//驱动插销油缸D10L-位移传感器	
				pos   := BYTE_TO_WORD(frame.data[5]) OR SHL(BYTE_TO_WORD(frame.data[6]),8);  	
				psPVDi^.arrPV[2].sNum[10].posVal.Current    := pos*0.1;	//驱动插销油缸D11L-位移传感器		
				pos   := BYTE_TO_WORD(frame.data[7]) OR SHL(BYTE_TO_WORD(frame.data[8]),8);  	
				psPVDi^.arrPV[2].sNum[11].posVal.Current   := pos*0.1;	//驱动插销油缸D12L-位移传感器		
				
			16#395:           //接收C9送来的数据
				pos   := BYTE_TO_WORD(frame.data[1]) OR SHL(BYTE_TO_WORD(frame.data[2]),8);  	
				psPVDi^.arrPV[1].sNum[8].posVal.Current  := pos*0.1;		//驱动插销油缸D00L2-位移传感器	
				pos   := BYTE_TO_WORD(frame.data[3]) OR SHL(BYTE_TO_WORD(frame.data[4]),8);  	
				psPVDi^.arrPV[1].sNum[1].posVal.Current  := pos*0.1;		//驱动插销油缸D00Q1-位移传感器	
				pos   := BYTE_TO_WORD(frame.data[5]) OR SHL(BYTE_TO_WORD(frame.data[6]),8);  	
				psPVDi^.arrPV[1].sNum[2].posVal.Current  := pos*0.1;		//驱动插销油缸D00Q2-位移传感器	
		END_CASE
	END_FOR


	gCan.C9RxCounter := gCan.C9RxMsg.RxCounter ;
END_IF

END_FUNCTION

// Device/Application/can/swmc_floor_rail/swmc_C10_Rx
FUNCTION swmc_C10_Rx : BOOL
VAR_INPUT
	CNT				: UINT;
	psYyz			: POINTER TO YyStation;
	
	psPVDi			: POINTER TO propValveModule_Di;
END_VAR
VAR
	frame	 	    : Can_baseframe;
	COB_ID			: UINT;
	I				: UINT;
	pos				: WORD;
END_VAR

IF gCan.C10RxMsg.RxCounter <>  gCan.C10RxCounter THEN    //接收到新的数据

	FOR  I := 1 TO  gCan.C10RxMsg.NoOfRxMessages DO
		frame :=CAN_Read_Data_SWMC(10,I);
		COB_ID :=	frame.id;    //获取ID
		CASE COB_ID OF     //根据ID解析协议
		//C10-0x3A0
			16#3A0:           //接收C10送来的数据
				pos := BYTE_TO_WORD(frame.data[1]) OR SHL(BYTE_TO_WORD(frame.data[2]),8);  	
				psPVDi^.arrPV[6].sNum[1].posVal.Current:= pos*0.1;	//驱动插销油缸D13Q-位移传感器	
				pos := BYTE_TO_WORD(frame.data[3]) OR SHL(BYTE_TO_WORD(frame.data[4]),8);  	
				psPVDi^.arrPV[6].sNum[2].posVal.Current:= pos*0.1;	//驱动插销油缸D14Q-位移传感器	
				pos := BYTE_TO_WORD(frame.data[5]) OR SHL(BYTE_TO_WORD(frame.data[6]),8);  	
				psPVDi^.arrPV[6].sNum[3].posVal.Current:= pos*0.1;	//驱动插销油缸D15Q-位移传感器		
				pos := BYTE_TO_WORD(frame.data[7]) OR SHL(BYTE_TO_WORD(frame.data[8]),8);  	
				psPVDi^.arrPV[6].sNum[4].posVal.Current:= pos*0.1;	//驱动插销油缸D16L1-位移传感器		
			//C10-0x3A1
			16#3A1:           //接收C10送来的数据
				pos := BYTE_TO_WORD(frame.data[1]) OR SHL(BYTE_TO_WORD(frame.data[2]),8);  	
				psPVDi^.arrPV[6].sNum[5].posVal.Current:= pos*0.1;	//驱动插销油缸D13L-位移传感器	
				pos := BYTE_TO_WORD(frame.data[3]) OR SHL(BYTE_TO_WORD(frame.data[4]),8);  	
				psPVDi^.arrPV[6].sNum[6].posVal.Current:= pos*0.1;	//驱动插销油缸D14L-位移传感器	
				pos := BYTE_TO_WORD(frame.data[5]) OR SHL(BYTE_TO_WORD(frame.data[6]),8);  	
				psPVDi^.arrPV[6].sNum[7].posVal.Current:= pos*0.1;	//驱动插销油缸D15L-位移传感器		
				pos := BYTE_TO_WORD(frame.data[7]) OR SHL(BYTE_TO_WORD(frame.data[8]),8);  	
				psPVDi^.arrPV[6].sNum[8].posVal.Current:= pos*0.1;	//驱动插销油缸D16L2-位移传感器
			
		END_CASE
	END_FOR


	gCan.C10RxCounter := gCan.C10RxMsg.RxCounter ;
END_IF

END_FUNCTION

// Device/Application/public_datum/yy_station/yysInterface
PROGRAM yysInterface
VAR
	
END_VAR

yysInterface_Status();

yysInterface_Cmd
(
	ADR(gImple.hydraPresStation),		//液压站地址
	gUI.cmdInverterFan,					//变频器风机
	gUI.cmdOilPumpFan,					//油泵风机
	gUI.cmdOilPumpM,					//油泵电机
	gUI.cmdOilPrePercent,				//油压百分比
	gUI.cmdOilPre_EN					//油压使能
);

ACTION yysInterface_Status:
	//压力
	gUI.arrStationPressure[1]:=gImple.hydraPresStation.Status.pressureStatus;	 		//压力传感器SQ1P(压力开关S1)
	gUI.arrStationPressure[2]:=gImple.hydraPresStation.Status.pressureV2;				//压力传感器SQ2P
	gUI.arrStationPressure[3]:=gImple.hydraPresStation.Status.pressureV3;				//压力传感器SQ3P
	gUI.arrStationPressure[4]:=gImple.hydraPresStation.Status.pressureV4;				//压力传感器SQ4P
	gUI.arrStationPressure[5]:=gImple.hydraPresStation.Status.pressureV5;				//压力传感器SQ5P	
	gUI.arrStationPressure[8]:=gImple.hydraPresStation.Status.pressureV8;				//压力传感器SQ8P
	gUI.arrStationPressure[9]:=gImple.hydraPresStation.Status.pressureV9;				//压力传感器SQ9P
	gUI.arrStationPressure[10]:=gImple.hydraPresStation.Status.pressureV10;				//压力传感器SQ10P
	gUI.arrStationPressure[11]:=gImple.hydraPresStation.Status.pressureV11;				//压力传感器SQ11P	
	
	//状态
	gUI.rTemperature:=gImple.hydraPresStation.Status.temperatureStatus;			//温度值
	gUI.bFluidLevel	:=gImple.hydraPresStation.Status.yeweiStatus;				//液位值
	
	gUI.bYysPower:=gImple.hydraPresStation.Status.HydraulicStation_Power;		//液压站上电
	gUI.bCtrlPower:=gImple.hydraPresStation.Status.Control_Power;				//控制电源上电
	gUI.bFreqConverterFan:=gImple.hydraPresStation.Status.InverterFan_Run;  	//变频风机启动
	gUI.bFreqConverter:=gImple.hydraPresStation.Status.FrequencyConversion_Run;	//变频器运行
	
	gUI.bOilPumpM_Fault:=gImple.hydraPresStation.Status.OilPumpM_Fault;			//油泵电机故障
	gUI.bOilPumpFan:=gImple.hydraPresStation.Status.OilPumpFan;					//油泵冷却风机-非故障
	gUI.bFreqConverter_Fault:=gImple.hydraPresStation.Status.FrequencyConversion_Fault;	//变频器故障
	gUI.bFreqConverterFan_Fault:=gImple.hydraPresStation.Status.InverterFan_Fault;		//变频器风机故障
END_ACTION

METHOD yysInterface_Cmd : BOOL
VAR_INPUT
	psYyz						:POINTER TO YyStation;
	cmdInverterFan				:BOOL;			//变频风机控制
	cmdOilPumpFan				:BOOL;    	    //油泵风机控制
	cmdOilPumpM					:BOOL;			//油泵电机控制
	cmdOilPrePercent			:REAL;			//油压控制
	cmdOilPre_EN				:BOOL;			//油压使能
END_VAR

VAR
	bSetCondition				:BOOL;			//温度、液位等状态要求
	wOilPrePercentTemp  		:WORD;
	wOilMaxPreVal				:WORD:=50;  	//最大限制为50
	
END_VAR

//液压站故障处理？

psYyz^.Cmd.HL_Mode_Ctrl:=0;				//高低速为0
psYyz^.Cmd.Energy_Swith:=0;				//储能开关为0
psYyz^.Cmd.OilPumpMotor_PN_Ctrl:=0;		//电机正反控制为0

//bSetCondition:=条件判定,满足后可执行以下动作
//IF bSetCondition 
//THEN

IF cmdOilPumpFan THEN					//油泵风扇控制
	psYyz^.Cmd.OilPumpFan_Ctrl:=1;
ELSE
	psYyz^.Cmd.OilPumpFan_Ctrl:=0;
END_IF

IF cmdInverterFan THEN					//变频器风扇控制
	psYyz^.Cmd.InverterFan_Ctrl:=1;
ELSE
	psYyz^.Cmd.InverterFan_Ctrl:=0;	
END_IF

IF cmdOilPumpFan THEN					//电机启动
	psYyz^.Cmd.OilPumpMotor_Ctrl:=1;
	psYyz^.Cmd.KEEP_Mode_Ctrl:=1;		//恒速模式
ELSE
	psYyz^.Cmd.OilPumpMotor_Ctrl:=0;
	psYyz^.Cmd.KEEP_Mode_Ctrl:=0;
END_IF

IF cmdOilPrePercent > wOilMaxPreVal THEN	//最大限制为 50%
	cmdOilPrePercent:=wOilMaxPreVal;
END_IF

IF cmdOilPre_EN THEN						//液压使能后才输出压力值
	wOilPrePercentTemp:=REAL_TO_WORD(cmdOilPrePercent*65535/100);
ELSE
	wOilPrePercentTemp:=0;
END_IF

psYyz^.Cmd.Oil_Pre_Val := wOilPrePercentTemp;
END_METHOD

END_PROGRAM

// Device/Application/can/old/swmc_C11_Rx
FUNCTION swmc_C11_Rx : BOOL
VAR_INPUT
	CNT				: UINT;
	psYyz			: POINTER TO YyStation;
	psPVTi			: POINTER TO propValveModule_Ti;
	
END_VAR
VAR
	frame	 	    : Can_baseframe;
	COB_ID			: UINT;
	I				: UINT;
	Pre				: UINT;
	pos				: WORD;
END_VAR

IF gCan.C11RxMsg.RxCounter <>  gCan.C11RxCounter THEN    //接收到新的数据

	FOR  I := 1 TO  gCan.C11RxMsg.NoOfRxMessages DO
		frame :=CAN_Read_Data_SWMC(11,I);
		COB_ID :=	frame.id;    //获取ID
		CASE COB_ID OF     //根据ID解析协议
		
		
			//C11-0x3B0
			16#3B0:           //接收C11送来的数据
				pos := BYTE_TO_WORD(frame.data[1]) OR SHL(BYTE_TO_WORD(frame.data[2]),8);  	
				psPVTi^.arrPV[1].sNum[1].posVal.Current:= pos*0.1;	
				pos := BYTE_TO_WORD(frame.data[3]) OR SHL(BYTE_TO_WORD(frame.data[4]),8);  
				psPVTi^.arrPV[1].sNum[2].posVal.Current:= pos*0.1;		
				pos := BYTE_TO_WORD(frame.data[5]) OR SHL(BYTE_TO_WORD(frame.data[6]),8);  
				psPVTi^.arrPV[1].sNum[3].posVal.Current:= pos*0.1;	
				pos := BYTE_TO_WORD(frame.data[7]) OR SHL(BYTE_TO_WORD(frame.data[8]),8);  	
				psPVTi^.arrPV[1].sNum[4].posVal.Current:= pos*0.1;

			//C6-0x3B1
			16#3B1:           //接收C11送来的数据
				pos := BYTE_TO_WORD(frame.data[1]) OR SHL(BYTE_TO_WORD(frame.data[2]),8);  	
				psPVTi^.arrPV[1].sNum[5].posVal.Current:= pos*0.1;	
				pos := BYTE_TO_WORD(frame.data[3]) OR SHL(BYTE_TO_WORD(frame.data[4]),8);  	
				psPVTi^.arrPV[1].sNum[6].posVal.Current:= pos*0.1;	
				pos := BYTE_TO_WORD(frame.data[5]) OR SHL(BYTE_TO_WORD(frame.data[6]),8);  	
				psPVTi^.arrPV[1].sNum[7].posVal.Current:= pos*0.1;	
				pos := BYTE_TO_WORD(frame.data[7]) OR SHL(BYTE_TO_WORD(frame.data[8]),8);  	
				psPVTi^.arrPV[1].sNum[8].posVal.Current:= pos*0.1;
			//C6-0x3B2
			16#3B2:           //接收C11送来的数据
				pos := BYTE_TO_WORD(frame.data[1]) OR SHL(BYTE_TO_WORD(frame.data[2]),8);  	
				psPVTi^.arrPV[1].sNum[9].posVal.Current:= pos*0.1;	
				pos := BYTE_TO_WORD(frame.data[3]) OR SHL(BYTE_TO_WORD(frame.data[4]),8);  	
				psPVTi^.arrPV[2].sNum[1].posVal.Current:= pos*0.1;		
				pos := BYTE_TO_WORD(frame.data[5]) OR SHL(BYTE_TO_WORD(frame.data[6]),8);  	
				psPVTi^.arrPV[2].sNum[2].posVal.Current:= pos*0.1;		
				pos := BYTE_TO_WORD(frame.data[7]) OR SHL(BYTE_TO_WORD(frame.data[8]),8);  	
				psPVTi^.arrPV[2].sNum[3].posVal.Current:= pos*0.1;	
			//C6-0x3B3
			16#3B3:           //接收C11送来的数据
				pos := BYTE_TO_WORD(frame.data[1]) OR SHL(BYTE_TO_WORD(frame.data[2]),8);  	
				psPVTi^.arrPV[2].sNum[4].posVal.Current:= pos*0.1;		
				pos := BYTE_TO_WORD(frame.data[3]) OR SHL(BYTE_TO_WORD(frame.data[4]),8);  	
				psPVTi^.arrPV[2].sNum[5].posVal.Current:= pos*0.1;		
				pos := BYTE_TO_WORD(frame.data[5]) OR SHL(BYTE_TO_WORD(frame.data[6]),8);  	
				psPVTi^.arrPV[2].sNum[6].posVal.Current:= pos*0.1;		
				pos := BYTE_TO_WORD(frame.data[7]) OR SHL(BYTE_TO_WORD(frame.data[8]),8);  	
				psPVTi^.arrPV[2].sNum[7].posVal.Current:= pos*0.1;	
			//C6-0x3B4
			16#3B4:           //接收C11送来的数据
				pos := BYTE_TO_WORD(frame.data[1]) OR SHL(BYTE_TO_WORD(frame.data[2]),8);  	
				psPVTi^.arrPV[2].sNum[8].posVal.Current:= pos*0.1;		
				pos := BYTE_TO_WORD(frame.data[3]) OR SHL(BYTE_TO_WORD(frame.data[4]),8);  	
				psPVTi^.arrPV[2].sNum[9].posVal.Current:= pos*0.1;		
				pos := BYTE_TO_WORD(frame.data[5]) OR SHL(BYTE_TO_WORD(frame.data[6]),8);  	
				psPVTi^.arrPV[2].sNum[10].posVal.Current:= pos*0.1;		
				pos := BYTE_TO_WORD(frame.data[7]) OR SHL(BYTE_TO_WORD(frame.data[8]),8);  	
				psPVTi^.arrPV[2].sNum[11].posVal.Current:= pos*0.1;	
			
		END_CASE
	END_FOR
	gCan.C11RxCounter := gCan.C11RxMsg.RxCounter ;
END_IF

END_FUNCTION

// Device/Application/can/old/CAN_COM
PROGRAM CAN_COM
VAR
	T_CNT   :UINT;

END_VAR

T_CNT := T_CNT+1;
IF  T_CNT > 1000 THEN
	 T_CNT := 1;
END_IF

swmc_C00_RX(T_CNT, ADR(gImple.hydraPresStation));
swmc_C00_TX(T_CNT, ADR(gImple.hydraPresStation));


swmc_C01_Rx(T_CNT,ADR(gImple.hydraPresStation),ADR(gImple.PV_GroupDi));
swmc_C01_Tx(T_CNT,ADR(gImple.PV_GroupDi));
swmc_C02_Rx(T_CNT,ADR(gImple.hydraPresStation),ADR(gImple.PV_GroupDi));
swmc_C02_Tx(T_CNT,ADR(gImple.PV_GroupDi));
swmc_C09_Rx(T_CNT,ADR(gImple.hydraPresStation),ADR(gImple.PV_GroupDi));
swmc_C10_Rx(T_CNT,ADR(gImple.hydraPresStation),ADR(gImple.PV_GroupDi));
	

swmc_C05_Rx(T_CNT,ADR(gImple.hydraPresStation),ADR(gImple.PV_GroupTi));
swmc_C05_Tx(T_CNT,ADR(gImple.PV_GroupTi));
swmc_C06_Rxold(T_CNT,ADR(gImple.hydraPresStation),ADR(gImple.PV_GroupTi));
swmc_C06_Tx(T_CNT,ADR(gImple.PV_GroupTi));
swmc_C11_Rx(T_CNT,ADR(gImple.hydraPresStation),ADR(gImple.PV_GroupTi));
swmc_C12_Rx(T_CNT,ADR(gImple.PV_GroupTi));

END_PROGRAM

// Device/Application/can/old/swmc_C06_Rxold
FUNCTION swmc_C06_Rxold : BOOL
VAR_INPUT
	CNT				: UINT;
	psYyz			: POINTER TO YyStation;
	psPVTi			: POINTER TO propValveModule_Ti;

END_VAR
VAR
	frame	 	    : Can_baseframe;
	COB_ID			: UINT;
	I				: UINT;
	Pre				: UINT;
	pos				: WORD;
END_VAR

IF gCan.C6RxMsg.RxCounter <>  gCan.C6RxCounter THEN    //接收到新的数据

	FOR  I := 1 TO  gCan.C6RxMsg.NoOfRxMessages DO
		frame :=CAN_Read_Data_SWMC(6,I);
		COB_ID :=	frame.id;    //获取ID
		CASE COB_ID OF     //根据ID解析协议
		
		
			//C6-0x360
			16#360:           //接收C6送来的数据
				pos := BYTE_TO_WORD(frame.data[1]) OR SHL(BYTE_TO_WORD(frame.data[2]),8);  	
				psPVTi^.arrPV[7].sNum[1].posVal.Current:= pos*0.1;	
				pos := BYTE_TO_WORD(frame.data[3]) OR SHL(BYTE_TO_WORD(frame.data[4]),8);  
				psPVTi^.arrPV[7].sNum[2].posVal.Current:= pos*0.1;		
				pos := BYTE_TO_WORD(frame.data[5]) OR SHL(BYTE_TO_WORD(frame.data[6]),8);  
				psPVTi^.arrPV[7].sNum[3].posVal.Current:= pos*0.1;	
				pos := BYTE_TO_WORD(frame.data[7]) OR SHL(BYTE_TO_WORD(frame.data[8]),8);  	
				psPVTi^.arrPV[7].sNum[4].posVal.Current:= pos*0.1;

			//C6-0x361
			16#361:           //接收C6送来的数据
				pos := BYTE_TO_WORD(frame.data[1]) OR SHL(BYTE_TO_WORD(frame.data[2]),8);  	
				psPVTi^.arrPV[7].sNum[5].posVal.Current:= pos*0.1;	
				pos := BYTE_TO_WORD(frame.data[3]) OR SHL(BYTE_TO_WORD(frame.data[4]),8);  	
				psPVTi^.arrPV[7].sNum[6].posVal.Current:= pos*0.1;	
				pos := BYTE_TO_WORD(frame.data[5]) OR SHL(BYTE_TO_WORD(frame.data[6]),8);  	
				psPVTi^.arrPV[7].sNum[7].posVal.Current:= pos*0.1;	
				pos := BYTE_TO_WORD(frame.data[7]) OR SHL(BYTE_TO_WORD(frame.data[8]),8);  	
				psPVTi^.arrPV[7].sNum[8].posVal.Current:= pos*0.1;
			//C6-0x362
			16#362:           //接收C6送来的数据
				pos := BYTE_TO_WORD(frame.data[1]) OR SHL(BYTE_TO_WORD(frame.data[2]),8);  	
				psPVTi^.arrPV[7].sNum[9].posVal.Current:= pos*0.1;	
				pos := BYTE_TO_WORD(frame.data[3]) OR SHL(BYTE_TO_WORD(frame.data[4]),8);  	
				psPVTi^.arrPV[7].sNum[10].posVal.Current:= pos*0.1;		
				pos := BYTE_TO_WORD(frame.data[5]) OR SHL(BYTE_TO_WORD(frame.data[6]),8);  	
				psPVTi^.arrPV[7].sNum[11].posVal.Current:= pos*0.1;		
				pos := BYTE_TO_WORD(frame.data[7]) OR SHL(BYTE_TO_WORD(frame.data[8]),8);  	
				psPVTi^.arrPV[7].sNum[12].posVal.Current:= pos*0.1;	
			//C6-0x363
			16#363:           //接收C6送来的数据
				pos := BYTE_TO_WORD(frame.data[1]) OR SHL(BYTE_TO_WORD(frame.data[2]),8);  	
				psPVTi^.arrPV[7].sNum[13].posVal.Current:= pos*0.1;		
				pos := BYTE_TO_WORD(frame.data[3]) OR SHL(BYTE_TO_WORD(frame.data[4]),8);  	
				psPVTi^.arrPV[7].sNum[14].posVal.Current:= pos*0.1;		
				pos := BYTE_TO_WORD(frame.data[5]) OR SHL(BYTE_TO_WORD(frame.data[6]),8);  	
				psPVTi^.arrPV[7].sNum[15].posVal.Current:= pos*0.1;		
				pos := BYTE_TO_WORD(frame.data[7]) OR SHL(BYTE_TO_WORD(frame.data[8]),8);  	
				psPVTi^.arrPV[7].sNum[16].posVal.Current:= pos*0.1;	
			//C6-0x364
			16#364:           //接收C6送来的数据
				pos := BYTE_TO_WORD(frame.data[1]) OR SHL(BYTE_TO_WORD(frame.data[2]),8);  	
				psPVTi^.arrPV[7].sNum[17].posVal.Current:= pos*0.1;		
				pos := BYTE_TO_WORD(frame.data[3]) OR SHL(BYTE_TO_WORD(frame.data[4]),8);  	
				psPVTi^.arrPV[7].sNum[18].posVal.Current:= pos*0.1;		
				pos := BYTE_TO_WORD(frame.data[5]) OR SHL(BYTE_TO_WORD(frame.data[6]),8);  	
				psPVTi^.arrPV[7].sNum[19].posVal.Current:= pos*0.1;		
				pos := BYTE_TO_WORD(frame.data[7]) OR SHL(BYTE_TO_WORD(frame.data[8]),8);  	
				psPVTi^.arrPV[7].sNum[20].posVal.Current:= pos*0.1;	
			//C6-0x365
			16#365:           //接收C6送来的数据
				pos := BYTE_TO_WORD(frame.data[1]) OR SHL(BYTE_TO_WORD(frame.data[2]),8);  	
				psPVTi^.arrPV[7].sNum[21].posVal.Current:= pos*0.1;		
				pos := BYTE_TO_WORD(frame.data[3]) OR SHL(BYTE_TO_WORD(frame.data[4]),8);  	
				psPVTi^.arrPV[7].sNum[22].posVal.Current:= pos*0.1;		
				pos := BYTE_TO_WORD(frame.data[5]) OR SHL(BYTE_TO_WORD(frame.data[6]),8);  	
				psPVTi^.arrPV[7].sNum[23].posVal.Current:= pos*0.1;		
				
				
				
			//C6-0x366
			16#366:           //接收C6送来的数据
				Pre :=BYTE_TO_WORD(frame.data[1]) OR SHL(BYTE_TO_WORD(frame.data[2]),8);
	 			psYyz^.Status.pressureV10:= 	(Pre-4000)/16000.0*400;	
				Pre :=BYTE_TO_WORD(frame.data[3]) OR SHL(BYTE_TO_WORD(frame.data[4]),8);
	 			psYyz^.Status.pressureV11:= 	(Pre-4000)/16000.0*400;	
			
	
			//C6.1 IO-0x367
			16#367:
				gImple.hydraPresStation.Status.arrSL[1]:=frame.data[1].0;	//限位开关SL1
				gImple.hydraPresStation.Status.arrSL[2]:=frame.data[1].1;	//限位开关SL2
		END_CASE
	END_FOR
	gCan.C6RxCounter := gCan.C6RxMsg.RxCounter ;
END_IF

END_FUNCTION

// Device/Application/can/old/swmc_C03_Rxl
FUNCTION swmc_C03_Rxl : BOOL
VAR_INPUT
	CNT				: UINT;
	psPVDi			: POINTER TO propValveModule_Di;
	psPVTi			: POINTER TO propValveModule_Ti;
END_VAR
VAR
	frame	 	    : Can_baseframe;
	COB_ID			: UINT;
	I				: UINT;
	pos				: WORD;
END_VAR

IF gCan.C3RxMsg.RxCounter <>  gCan.C3RxCounter THEN    //接收到新的数据

	FOR  I := 1 TO  gCan.C3RxMsg.NoOfRxMessages DO
		frame :=CAN_Read_Data_SWMC(3,I);
		COB_ID :=	frame.id;    //获取ID
		CASE COB_ID OF     //根据ID解析协议
	
			//C3-0x330
			16#330:           //接收C3送来的数据
				pos := BYTE_TO_WORD(frame.data[1]) OR SHL(BYTE_TO_WORD(frame.data[2]),8);  	
				psPVTi^.arrRotSYN[31].sNum[1].posVal.Current:= pos*0.1;	//天-驱动插销油缸E31Q-位移传感器		
				pos := BYTE_TO_WORD(frame.data[3]) OR SHL(BYTE_TO_WORD(frame.data[4]),8);  	
				psPVTi^.arrRotSYN[31].sNum[2].posVal.Current:= pos*0.1;	//天-驱动插销油缸E31Q1-位移传感器	
				pos := BYTE_TO_WORD(frame.data[5]) OR SHL(BYTE_TO_WORD(frame.data[6]),8);  	
				psPVDi^.arrRotSYN[31].sNum[1].posVal.Current:= pos*0.1;	//地-驱动插销油缸D31Q-位移传感器	
				pos := BYTE_TO_WORD(frame.data[7]) OR SHL(BYTE_TO_WORD(frame.data[8]),8);  	
				psPVDi^.arrRotSYN[31].sNum[2].posVal.Current:= pos*0.1;	//地-驱动插销油缸D31Q1-位移传感器	
			//C3-0x331
			16#331:           //接收C3送来的数据
				pos := BYTE_TO_WORD(frame.data[1]) OR SHL(BYTE_TO_WORD(frame.data[2]),8);  	
				psPVDi^.arrRotSYN[31].sNum[3].posVal.Current:= pos*0.1;	//地-驱动插销油缸D31Q2-位移传感器	
	
				
		END_CASE
	END_FOR


	gCan.C3RxCounter := gCan.C3RxMsg.RxCounter ;
END_IF

END_FUNCTION

// Device/Application/can/old/swmc_C04_Rxl
FUNCTION swmc_C04_Rxl : BOOL
VAR_INPUT
	CNT				: UINT;
	psPVDi			: POINTER TO propValveModule_Di;
	psPVTi			: POINTER TO propValveModule_Ti;
END_VAR
VAR
	frame	 	    : Can_baseframe;
	COB_ID			: UINT;
	I				: UINT;
	pos				: WORD;
END_VAR

IF gCan.C4RxMsg.RxCounter <>  gCan.C4RxCounter THEN    //接收到新的数据

	FOR  I := 1 TO  gCan.C4RxMsg.NoOfRxMessages DO
		frame :=CAN_Read_Data_SWMC(4,I);
		COB_ID :=	frame.id;    //获取ID
		CASE COB_ID OF     //根据ID解析协议
	
			//C3-0x340
			16#340:           //接收C3送来的数据
				pos := BYTE_TO_WORD(frame.data[1]) OR SHL(BYTE_TO_WORD(frame.data[2]),8);  	
				psPVTi^.arrRotSYN[32].sNum[1].posVal.Current:= pos*0.1;	//天-驱动插销油缸E32Q-位移传感器			
				pos := BYTE_TO_WORD(frame.data[3]) OR SHL(BYTE_TO_WORD(frame.data[4]),8);  	
				psPVTi^.arrRotSYN[32].sNum[2].posVal.Current:= pos*0.1;	//天-驱动插销油缸E32Q1-位移传感器	
				pos := BYTE_TO_WORD(frame.data[5]) OR SHL(BYTE_TO_WORD(frame.data[6]),8);  	
				psPVDi^.arrRotSYN[32].sNum[1].posVal.Current:= pos*0.1;	//地-驱动插销油缸D32Q-位移传感器	
				pos := BYTE_TO_WORD(frame.data[7]) OR SHL(BYTE_TO_WORD(frame.data[8]),8);  	
				psPVDi^.arrRotSYN[32].sNum[2].posVal.Current:= pos*0.1;	//地-驱动插销油缸D32Q1-位移传感器	
			//C3-0x341
			16#341:           //接收C3送来的数据
				pos := BYTE_TO_WORD(frame.data[1]) OR SHL(BYTE_TO_WORD(frame.data[2]),8);  	
				psPVDi^.arrRotSYN[32].sNum[3].posVal.Current:= pos*0.1;	//地-驱动插销油缸D32Q2-位移传感器	
	
				
		END_CASE
	END_FOR


	gCan.C4RxCounter := gCan.C4RxMsg.RxCounter ;
END_IF

END_FUNCTION

// Device/Application/can/old/swmc_C03_Txl
FUNCTION swmc_C03_Txl : BOOL
VAR_INPUT
	CNT				: UINT;
	
	psPVDi			: POINTER TO propValveModule_Di;
	psPVTi			: POINTER TO propValveModule_Ti;

END_VAR
VAR
	senddata	: ARRAY[1..8] OF BYTE;
	Send_cnt	: UINT;
END_VAR

//速度控制--待定
Send_cnt :=  CNT MOD 3;

CASE Send_cnt OF
	
	1:
 	//C3-0x430
	senddata[1] :=  WORD_TO_BYTE(psPVTi^.arrRotSYN[31].arrPercVal[1]);  		 //驱动油缸电比例阀DTE31Q1	
	senddata[2] :=  WORD_TO_BYTE(SHR(psPVTi^.arrRotSYN[31].arrPercVal[1],8));    //0-65535  对应0-100  

	senddata[3] :=  WORD_TO_BYTE(psPVTi^.arrRotSYN[31].arrPercVal[2]);  		   //驱动油缸电比例阀DTE31Q2
	senddata[4] :=  WORD_TO_BYTE(SHR(psPVTi^.arrRotSYN[31].arrPercVal[2],8));    //0-65535  对应0-100  
	
	senddata[5] :=  WORD_TO_BYTE(psPVTi^.arrRotSYN[31].arrPercVal[3]);  		   //驱动油缸电比例阀DTE31Q3	
	senddata[6] :=  WORD_TO_BYTE(SHR(psPVTi^.arrRotSYN[31].arrPercVal[3],8));    //0-65535  对应0-100  

	senddata[7] :=  WORD_TO_BYTE(psPVTi^.arrRotSYN[31].arrPercVal[4]);  		   //驱动油缸电比例阀DTE31Q4
	senddata[8] :=  WORD_TO_BYTE(SHR(psPVTi^.arrRotSYN[31].arrPercVal[4],8));    //0-65535  对应0-100  

	
	//发送至C3
	CAN_Send_Data_SWMC(3, 16#430,senddata);				//发送ID 0x430到C3
	
	2:
 	//C3-0x431
	senddata[1] :=  WORD_TO_BYTE(psPVDi^.arrRotSYN[31].arrPercVal[1]);  		   //驱动油缸电比例阀DTD31Q1	
	senddata[2] :=  WORD_TO_BYTE(SHR(psPVDi^.arrRotSYN[31].arrPercVal[1],8));    //0-65535  对应0-100  

	senddata[3] :=  WORD_TO_BYTE(psPVDi^.arrRotSYN[31].arrPercVal[2]);  		   //驱动油缸电比例阀DTD31Q1
	senddata[4] :=  WORD_TO_BYTE(SHR(psPVDi^.arrRotSYN[31].arrPercVal[2],8));    //0-65535  对应0-100  
	
	senddata[5] :=  WORD_TO_BYTE(psPVDi^.arrRotSYN[31].arrPercVal[3]);  		   //驱动油缸电比例阀DTD31Q3	
	senddata[6] :=  WORD_TO_BYTE(SHR(psPVDi^.arrRotSYN[31].arrPercVal[3],8));    //0-65535  对应0-100  

	senddata[7] :=  WORD_TO_BYTE(psPVDi^.arrRotSYN[31].arrPercVal[4]);  		   //驱动油缸电比例阀DTD31Q3
	senddata[8] :=  WORD_TO_BYTE(SHR(psPVDi^.arrRotSYN[31].arrPercVal[4],8));    //0-65535  对应0-100  
	
	
	//发送至C3
	CAN_Send_Data_SWMC(3, 16#431,senddata);				//发送ID 0x430到C3
	
	
END_CASE

END_FUNCTION

// Device/Application/can/old/swmc_C04_Txl
FUNCTION swmc_C04_Txl : BOOL
VAR_INPUT
	CNT				: UINT;
	
	psPVDi			: POINTER TO propValveModule_Di;
	psPVTi			: POINTER TO propValveModule_Ti;

END_VAR
VAR
	senddata	: ARRAY[1..8] OF BYTE;
	Send_cnt	: UINT;
END_VAR

//速度控制--待定
Send_cnt :=  CNT MOD 3;

CASE Send_cnt OF
	
	1:
 	//C4-0x440
	senddata[1] :=  WORD_TO_BYTE(psPVTi^.arrRotSYN[32].arrPercVal[1]);  		   //驱动油缸电比例阀DTE31Q1	
	senddata[2] :=  WORD_TO_BYTE(SHR(psPVTi^.arrRotSYN[32].arrPercVal[1],8));    //0-65535  对应0-100  

	senddata[3] :=  WORD_TO_BYTE(psPVTi^.arrRotSYN[32].arrPercVal[2]);  		   //驱动油缸电比例阀DTE31Q2
	senddata[4] :=  WORD_TO_BYTE(SHR(psPVTi^.arrRotSYN[32].arrPercVal[2],8));    //0-65535  对应0-100  
	
	senddata[5] :=  WORD_TO_BYTE(psPVTi^.arrRotSYN[32].arrPercVal[3]);  		   //驱动油缸电比例阀DTE31Q3	
	senddata[6] :=  WORD_TO_BYTE(SHR(psPVTi^.arrRotSYN[32].arrPercVal[3],8));    //0-65535  对应0-100  

	senddata[7] :=  WORD_TO_BYTE(psPVTi^.arrRotSYN[32].arrPercVal[4]);  		   //驱动油缸电比例阀DTE31Q4
	senddata[8] :=  WORD_TO_BYTE(SHR(psPVTi^.arrRotSYN[32].arrPercVal[4],8));    //0-65535  对应0-100  

	
	//发送至C4
	CAN_Send_Data_SWMC(4, 16#440,senddata);				//发送ID 0x440到C4
	
	2:
 	//C4-0x441
	senddata[1] :=  WORD_TO_BYTE(psPVDi^.arrRotSYN[32].arrPercVal[1]);  		   //驱动油缸电比例阀DTD31Q1	
	senddata[2] :=  WORD_TO_BYTE(SHR(psPVDi^.arrRotSYN[32].arrPercVal[1],8));    //0-65535  对应0-100  

	senddata[3] :=  WORD_TO_BYTE(psPVDi^.arrRotSYN[32].arrPercVal[2]);  		   //驱动油缸电比例阀DTD31Q1
	senddata[4] :=  WORD_TO_BYTE(SHR(psPVDi^.arrRotSYN[32].arrPercVal[2],8));    //0-65535  对应0-100  
	
	senddata[5] :=  WORD_TO_BYTE(psPVDi^.arrRotSYN[32].arrPercVal[3]);  		   //驱动油缸电比例阀DTD31Q3	
	senddata[6] :=  WORD_TO_BYTE(SHR(psPVDi^.arrRotSYN[32].arrPercVal[3],8));    //0-65535  对应0-100  

	senddata[7] :=  WORD_TO_BYTE(psPVDi^.arrRotSYN[32].arrPercVal[4]);  		   //驱动油缸电比例阀DTD31Q3
	senddata[8] :=  WORD_TO_BYTE(SHR(psPVDi^.arrRotSYN[32].arrPercVal[4],8));    //0-65535  对应0-100  
	
	
	//发送至C4
	CAN_Send_Data_SWMC(4, 16#441,senddata);				//发送ID 0x440到C4
	
	
END_CASE

END_FUNCTION

// Device/Application/public_datum/otherContent/PB_Pos_Check
FUNCTION_BLOCK PB_Pos_Check
VAR_INPUT
	Extend_Pos		:REAL;			//伸出位置
	Retract_Pos		:REAL;			//收回位置
	Act_Pos			:REAL;			//当前位置
	Err				:REAL;			//误差范围
END_VAR
VAR_OUTPUT
	S_Out		:POS_Status;		//输出状态
END_VAR
VAR
	E_cnt			:UINT:=0;			//伸出检测计数
	R_cnt			:UINT:=0;			//收回检测计数
	C_Out			:POS_Status;		//输出状态
END_VAR

// 10 ms 调用1次

// 开始检测
IF Act_Pos > 1 THEN    //实际位置总是大于1mm的
	IF   (Act_Pos  >= Extend_Pos -Err) THEN    //满足伸出误差
		E_cnt := E_cnt+1;
		R_cnt :=0;
	ELSIF  Act_Pos <=  (Retract_Pos+ Err) THEN	  //满足收回误差
		R_cnt := R_cnt+1;
		E_cnt := 0;
	ELSE
	   E_cnt := 0;
	   R_cnt :=0;
	END_IF
	IF  E_cnt >= 10 THEN    //是否为伸出状态
		E_cnt := 10;
		C_Out := POS_Status.enum_Extend;
	ELSIF  R_cnt >=10 THEN		//是否为收回状态
		R_cnt := 10;
		C_Out := POS_Status.enum_Retract;
	ELSE
		C_Out := POS_Status.enum_Run;
	END_IF
ELSE		//状态未知
  E_cnt := 0;
  R_cnt :=0;
  C_Out :=  POS_Status.enum_UNKOWN;  	
END_IF

S_Out :=  C_Out;

END_FUNCTION_BLOCK

// Device/Application/public_datum/otherContent/posCheckUnit
FUNCTION posCheckUnit : POS_Status
VAR_INPUT
	Extend_Pos		:REAL;			//伸出位置
	Retract_Pos		:REAL;			//收回位置
	Act_Pos			:REAL;			//当前位置
	Err				:REAL;			//误差范围
END_VAR
VAR
	E_cnt			:UINT:=0;			//伸出检测计数
	R_cnt			:UINT:=0;			//收回检测计数
	C_Out			:POS_Status;		//输出状态
END_VAR

// 10 ms 调用1次

// 开始检测
IF Act_Pos > 1 THEN    //实际位置总是大于1mm的
	IF   (Act_Pos  >= Extend_Pos -Err) THEN    //满足伸出误差
		E_cnt := E_cnt+1;
		R_cnt :=0;
	ELSIF  Act_Pos <=  (Retract_Pos+ Err) THEN	  //满足收回误差
		R_cnt := R_cnt+1;
		E_cnt := 0;
	ELSE
	   E_cnt := 0;
	   R_cnt :=0;
	END_IF
	IF  E_cnt >= 10 THEN    //是否为伸出状态
		E_cnt := 10;
		C_Out := POS_Status.enum_Extend;
	ELSIF  R_cnt >=10 THEN		//是否为收回状态
		R_cnt := 10;
		C_Out := POS_Status.enum_Retract;
	ELSE
		C_Out := POS_Status.enum_Run;
	END_IF
ELSE		//状态未知
	E_cnt := 0;
  	R_cnt := 0;
 	C_Out :=  POS_Status.enum_UNKOWN;  	
END_IF

posCheckUnit :=  C_Out;

END_FUNCTION

// Device/Application/public_datum/otherContent/SP_CC_YK_Run_BCtrl
FUNCTION_BLOCK SP_CC_YK_Run_BCtrl
VAR_INPUT
	Run			:Ctrl_Status1;
	Sensor1		:Sensor_Info;
	Sensor2		:Sensor_Info;
	Param1		:POS_Param;
	Param2		:POS_Param;
END_VAR
VAR_OUTPUT
	E_Ctrl		:BOOL;			//伸出
	R_Ctrl		:BOOL;			//收回
	Status		:POS_Status;	//位置状态
	Err_OUT		:BOOL;			//错误输出
END_VAR
VAR
	POS1C		:PB_Pos_Check;
	POS2C		:PB_Pos_Check;
	Ctrl_Run	: Ctrl_Status1;
	Err_Cnt		: UINT;
END_VAR


POS1C(
	Extend_Pos:= Param1.Extend_pos , 
	Retract_Pos:= Param1.Retract_pos, 
	Act_Pos:= Sensor1.POS, 
	Err:= 2.0, 
	S_Out=> );		//传感器位置检测
POS2C(
	Extend_Pos:= Param2.Extend_pos , 
	Retract_Pos:= Param2.Retract_pos, 
	Act_Pos:= Sensor2.POS, 
	Err:= 2.0, 
	S_Out=> );		//传感器位置检测



CASE   Run OF		//根据输入状态 进行运行
	Ctrl_Status1.Extend:
	    IF  (POS1C.S_Out <> POS_Status.enum_Extend)OR (POS2C.S_Out <>  POS_Status.enum_Extend) THEN		//位置不是伸出位置
			IF  Ctrl_Run <> Ctrl_Status1.Extend_Run THEN		//不在伸出运行状态
				Err_Cnt := 0;
				Err_OUT := FALSE;
				Ctrl_Run := Ctrl_Status1.Extend_Run;
			END_IF
		END_IF
	Ctrl_Status1.Retract:
		IF  (POS1C.S_Out <> POS_Status.enum_Retract)OR (POS2C.S_Out <>  POS_Status.enum_Retract) THEN		//位置不是伸出位置
			IF  Ctrl_Run <> Ctrl_Status1.Retract_Run THEN		//不在伸出运行状态
				Err_Cnt := 0;
				Err_OUT := FALSE;
				Ctrl_Run := Ctrl_Status1.Retract_Run;
			END_IF
		END_IF
	Ctrl_Status1.Stop:
	    Err_Cnt := 0;
		Err_OUT := FALSE;
		Ctrl_Run := Ctrl_Status1.Stop;
	Ctrl_Status1.Free:
		
END_CASE

Err_Cnt := Err_Cnt +1;    //故障计数
CASE Ctrl_Run OF
	Ctrl_Status1.Extend_Run:		//伸出运行
		 IF  (POS1C.S_Out = POS_Status.enum_Extend)AND (POS2C.S_Out =  POS_Status.enum_Extend) THEN	   //两个均伸出，关闭输出 进入空闲态
			E_Ctrl := 0;
			R_Ctrl := 0;
			Err_Cnt :=0;
			Ctrl_Run :=  Ctrl_Status1.Free;
		 ELSE		//继续伸出
			E_Ctrl := 1;
			R_Ctrl := 0; 
			IF  Err_Cnt > 30*100 THEN		//超时未伸出
				Ctrl_Run :=Ctrl_Status1.Err;  
			END_IF
		 END_IF
	Ctrl_Status1.Retract_Run:	//回收运行
		 IF  (POS1C.S_Out = POS_Status.enum_Retract)AND (POS2C.S_Out =  POS_Status.enum_Retract) THEN	   //两个均收回，关闭输出 进入空闲态
			E_Ctrl := 0;
			R_Ctrl := 0;
			Err_Cnt :=0;
			Ctrl_Run :=  Ctrl_Status1.Free;
		 ELSE		//继续收回
			E_Ctrl := 0;
			R_Ctrl := 1; 
			IF  Err_Cnt > 30*100 THEN		//超时未收回
				Ctrl_Run :=Ctrl_Status1.Err;  
			END_IF
		 END_IF
	Ctrl_Status1.Stop:
		E_Ctrl := 0;
		R_Ctrl := 0;
		Err_Cnt := 0;
	Ctrl_Status1.Free:
		E_Ctrl := 0;
		R_Ctrl := 0;
		Err_Cnt := 0;
	Ctrl_Status1.Err:
		Err_Cnt := 0;
		E_Ctrl := 0;
		R_Ctrl := 0;
		Err_OUT := TRUE;    // 错误输出
END_CASE

//根据两个位置传感器状态 输出状态

IF  Ctrl_Run = Ctrl_Status1.Err OR  POS1C.S_Out = POS_Status.enum_UNKOWN OR  POS2C.S_Out = POS_Status.enum_UNKOWN   THEN		//出错或者有个状态为未知
	Status := POS_Status.enum_UNKOWN;
ELSIF  (POS1C.S_Out = POS_Status.enum_Retract)AND (POS2C.S_Out =  POS_Status.enum_Retract) THEN		//收回状态
	Status := POS_Status.enum_Retract;
ELSIF (POS1C.S_Out = POS_Status.enum_Extend)AND (POS2C.S_Out =  POS_Status.enum_Extend) THEN		//伸出状态
	Status := POS_Status.enum_Extend;
ELSE		//运行状态
	Status := POS_Status.enum_Run;
END_IF

END_FUNCTION_BLOCK

// Device/Application/public_datum/otherContent/modbusold/modbusAct0
PROGRAM modbusAct0
VAR
	bInitialize				:BOOL:=TRUE;
	iClientConnect			:UINT:=1;
	iCountAct				:UINT:=10;
	iErrCode				:BYTE;
	iTemp					:UINT;
	fbModbusClient				: ModbusTcp_Client;
	fbReadHoldRegister  		: ReadHoldRegister;					//读保持寄存器
	fbWriteSingleHoldRegister	: WriteSingleHoldRegister;			//写保持1寄存器
	fbWriteMutiRegister			: WriteMutiRegister;				//写多个保持寄存器
END_VAR

IF bInitialize THEN
	initAddrPacket0(ADR(gModbus.master));
	bInitialize:=FALSE;
END_IF

IF iClientConnect<>1 THEN
	fbModbusClient(sIPAddress:='192.168.2.24',uiPort:=520);
END_IF

IF fbModbusClient.bSuccess THEN
	iClientConnect:=1;
	
	CASE iCountAct OF
		10:
			handleHeartbeat0();	//心跳
		20:
			handleCommand0();	//处理控制指令
		30:
			handleStatus0();	//发送油缸状态
		40:
			handlePosition0();	//发送位移传感器信息
	END_CASE
	
	
	
END_IF

METHOD PRIVATE getStatus0 : BOOL
VAR_INPUT
END_VAR
VAR
	iVT					:INT;
	iVT1				:INT;
	eTemp				:cmdStat;
	b0					:BYTE;
	b1					:BYTE;
	arrStatusPre		:ARRAY[11..77] OF USINT;
END_VAR
VAR CONSTANT
	aNo		:ARRAY [1..7] OF INT :=[6, 5,1,1,1,5, 7];		//每个比例阀下开关阀的数量(天轨):arrMappingRealNumTiG
END_VAR
FOR iVT:=1 TO 7 DO				//每个比例阀
	FOR iVT1:=1 TO aNo[iVT] DO	//比例阀中每个开关阀
		eTemp:=gImple.PV_GroupTi.arrPV[iVT].sColumn[iVT1].eStat;
		CASE eTemp OF
			cmdStat.eNormal:	//初始态
				arrStatusPre[iVT*10+iVT1]:= 0;
			cmdStat.Extend_Done://伸出
				arrStatusPre[iVT*10+iVT1]:= 1;
			cmdStat.eRun:		//运行
				arrStatusPre[iVT*10+iVT1]:= 2;
			cmdStat.Retract_Done://收回
				arrStatusPre[iVT*10+iVT1]:= 4;
			cmdStat.eError:
				arrStatusPre[iVT*10+iVT1]:= 15;
		END_CASE
	END_FOR	
END_FOR

b0 := arrStatusPre[13] OR SHL(arrStatusPre[16],4);
b1 := arrStatusPre[21] OR SHL(arrStatusPre[22],4);
gModbus.master.sStatus.arrDat[40] := b0 OR SHL(BYTE_TO_WORD(b1),8);

b0 := arrStatusPre[23] OR SHL(arrStatusPre[24],4);
b1 := arrStatusPre[25] OR SHL(arrStatusPre[64],4);
gModbus.master.sStatus.arrDat[41] := b0 OR SHL(BYTE_TO_WORD(b1),8);

b0 := arrStatusPre[63] OR SHL(arrStatusPre[65],4);
b1 := arrStatusPre[76] OR SHL(arrStatusPre[71],4);
gModbus.master.sStatus.arrDat[42] := b0 OR SHL(BYTE_TO_WORD(b1),8);

b0 := arrStatusPre[72] OR SHL(arrStatusPre[73],4);
b1 := arrStatusPre[77] OR SHL(arrStatusPre[11],4);
gModbus.master.sStatus.arrDat[43] := b0 OR SHL(BYTE_TO_WORD(b1),8);

b0 := arrStatusPre[12] OR SHL(arrStatusPre[31],4);
b1 := arrStatusPre[41] OR SHL(arrStatusPre[51],4);
gModbus.master.sStatus.arrDat[44] := b0 OR SHL(BYTE_TO_WORD(b1),8);

b0 := arrStatusPre[61] OR SHL(arrStatusPre[62],4);
b1 := arrStatusPre[74] OR SHL(arrStatusPre[75],4);
gModbus.master.sStatus.arrDat[45] := b0 OR SHL(BYTE_TO_WORD(b1),8);

b0 := arrStatusPre[15] OR SHL(arrStatusPre[14],4);
b1 := 0;
gModbus.master.sStatus.arrDat[46] := b0 OR SHL(BYTE_TO_WORD(b1),8);
END_METHOD

METHOD PRIVATE initAddrPacket0 : BOOL
VAR_INPUT
	pModbus			: POINTER TO ModbusStruct;
END_VAR
pModbus^.sHeartbeat.wStartAddr	:= 5;
pModbus^.sHeartbeat.wAmount		:= 1;

pModbus^.sCmd.wStartAddr		:= 20;
pModbus^.sCmd.wAmount			:= 4;

pModbus^.sStatus.wStartAddr		:= 40;
pModbus^.sStatus.wAmount		:= 7;

pModbus^.sPos.wStartAddr		:= 200;
pModbus^.sPos.wAmount			:= 75;
END_METHOD

ACTION handleHeartbeat0:
(*
fbReadHoldRegister(
	xExecute 	:= TRUE,
	slaveId		:= 1, 
	wStartAdr	:= gModbus.master.sHeartbeat.wStartAddr,
	wLen		:= gModbus.master.sHeartbeat.wAmount,  
	pTcpStream	:= fbModbusClient.pfbTcpStream,
	modbusHoldRegData:= gModbus.arrBufferDat);
	
IF fbReadHoldRegister.bSucced THEN
	fbReadHoldRegister(
		xExecute :=FALSE,
		modbusHoldRegData:= gModbus.arrBufferDat);
	gModbus.master.sHeartbeat.iHeartNum:=gModbus.arrBufferDat[gModbus.master.sHeartbeat.wStartAddr];
*)	
	
	fbWriteSingleHoldRegister(
		xExecute 	:=TRUE,
		slaveId 	:=1,
		setAddr		:=gModbus.master.sHeartbeat.wStartAddr,
		setvalue	:=gModbus.master.sHeartbeat.iHeartNum,
		pTcpStream	:=fbModbusClient.pfbTcpStream);
	IF fbWriteSingleHoldRegister.bSucced THEN
		fbWriteSingleHoldRegister(xExecute:=FALSE);
		gModbus.master.sHeartbeat.iHeartNum:=gModbus.master.sHeartbeat.iHeartNum+1;
		iCountAct :=20;	
	END_IF
	IF fbWriteSingleHoldRegister.berror THEN
		fbWriteSingleHoldRegister(xExecute:=FALSE);
		fbModbusClient.M_Reset();
		iCountAct:=10;
		iClientConnect:=0;
		iErrCode:=fbWriteSingleHoldRegister.errCode;
	END_IF
(*
END_IF

IF fbReadHoldRegister.berror THEN
	fbReadHoldRegister(
		xExecute :=FALSE,
		modbusHoldRegData:= gModbus.arrBufferDat);
	iCountAct:=10;	
	iErrCode:=fbReadHoldRegister.errCode;
END_IF
*)
END_ACTION

ACTION handlePosition0:

modbusAct0.getPos0();	//获取位置

fbWriteMutiRegister(
	xExecute	:=TRUE,
	slaveId		:=1,
	startAddr	:=gModbus.master.sPos.wStartAddr,
	wRegNum		:=gModbus.master.sPos.wAmount,
	value		:=ADR(gModbus.master.sPos.arrDat),
	pTcpStream	:=fbModbusClient.pfbTcpStream
	);
	
IF fbWriteMutiRegister.bSucced THEN
	fbWriteMutiRegister(xExecute:=FALSE);
	iCountAct:=10;
END_IF

IF fbWriteMutiRegister.berror THEN
	fbWriteMutiRegister(xExecute:=FALSE);
	fbModbusClient.M_Reset();
	iCountAct:=10;
	iClientConnect:=0;
	iErrCode :=fbWriteMutiRegister.errCode;
END_IF
END_ACTION

ACTION handleStatus0:

modbusAct.getStatus();	//获取状态

fbWriteMutiRegister(
	xExecute	:=TRUE,
	slaveId		:=1,
	startAddr	:=gModbus.master.sStatus.wStartAddr,
	wRegNum		:=gModbus.master.sStatus.wAmount,
	value		:=ADR(gModbus.master.sStatus.arrDat),
	pTcpStream	:=fbModbusClient.pfbTcpStream
	);
	
IF fbWriteMutiRegister.bSucced THEN
	fbWriteMutiRegister(xExecute:=FALSE);
	iCountAct:=40;
END_IF

IF fbWriteMutiRegister.berror THEN
	fbWriteMutiRegister(xExecute:=FALSE);
	fbModbusClient.M_Reset();
	iCountAct:=10;
	iClientConnect:=0;
	iErrCode :=fbWriteMutiRegister.errCode;
END_IF
END_ACTION

ACTION handleCommand0:
fbReadHoldRegister(
	xExecute	:=TRUE,
	slaveId		:=1,
	wStartAdr	:=gModbus.master.sCmd.wStartAddr,
	wLen		:=gModbus.master.sCmd.wAmount,
	pTcpStream	:= fbModbusClient.pfbTcpStream,
	modbusHoldRegData:= gModbus.arrBufferDat);

IF fbReadHoldRegister.bSucced THEN
	FOR iTemp:=0 TO 3 DO
		gModbus.master.sCmd.arrDat[20+iTemp]:=gModbus.arrBufferDat[gModbus.master.sCmd.wStartAddr+iTemp];	
	END_FOR	
	fbReadHoldRegister(
		xExecute := FALSE,
		modbusHoldRegData:=g_modbusHoldRegData);
	//执行控制指令
	modbusAct0.executeCmd0();
	iCountAct :=30;		

END_IF

IF fbReadHoldRegister.berror THEN
	fbReadHoldRegister(
		xExecute :=FALSE,
		modbusHoldRegData:= gModbus.arrBufferDat);
	iCountAct:=10;	
	iErrCode:=fbReadHoldRegister.errCode;
END_IF
END_ACTION

ACTION getPosA0:

END_ACTION

METHOD PRIVATE getPos0 : BOOL
VAR_INPUT
END_VAR
gModbus.master.sPos.arrDat[200]:= REAL_TO_WORD(gUI.TiG.arrPV[1].sNum[5].rPercent);	//E00L
gModbus.master.sPos.arrDat[201]:= REAL_TO_WORD(gUI.TiG.arrPV[1].sNum[9].rPercent);	//E01L

gModbus.master.sPos.arrDat[202]:= REAL_TO_WORD(gUI.TiG.arrPV[2].sNum[1].rPercent);	//E02L
gModbus.master.sPos.arrDat[203]:= REAL_TO_WORD(gUI.TiG.arrPV[2].sNum[2].rPercent);	//E03L
gModbus.master.sPos.arrDat[204]:= REAL_TO_WORD(gUI.TiG.arrPV[2].sNum[3].rPercent);	//E04L
gModbus.master.sPos.arrDat[205]:= REAL_TO_WORD(gUI.TiG.arrPV[2].sNum[4].rPercent);
gModbus.master.sPos.arrDat[206]:= REAL_TO_WORD(gUI.TiG.arrPV[2].sNum[5].rPercent);
gModbus.master.sPos.arrDat[207]:= REAL_TO_WORD(gUI.TiG.arrPV[2].sNum[6].rPercent);
gModbus.master.sPos.arrDat[208]:= REAL_TO_WORD(gUI.TiG.arrPV[2].sNum[7].rPercent);
gModbus.master.sPos.arrDat[209]:= REAL_TO_WORD(gUI.TiG.arrPV[2].sNum[8].rPercent);
gModbus.master.sPos.arrDat[210]:= REAL_TO_WORD(gUI.TiG.arrPV[2].sNum[9].rPercent);
gModbus.master.sPos.arrDat[211]:= REAL_TO_WORD(gUI.TiG.arrPV[2].sNum[10].rPercent);
gModbus.master.sPos.arrDat[212]:= REAL_TO_WORD(gUI.TiG.arrPV[2].sNum[11].rPercent);	//E12L

gModbus.master.sPos.arrDat[213]:= REAL_TO_WORD(gUI.TiG.arrPV[6].sNum[6].rPercent);	//E13L
gModbus.master.sPos.arrDat[214]:= REAL_TO_WORD(gUI.TiG.arrPV[6].sNum[4].rPercent);	//E14L
gModbus.master.sPos.arrDat[215]:= REAL_TO_WORD(gUI.TiG.arrPV[6].sNum[5].rPercent);	//E15L
gModbus.master.sPos.arrDat[216]:= REAL_TO_WORD(gUI.TiG.arrPV[6].sNum[7].rPercent);	//E16L1
gModbus.master.sPos.arrDat[217]:= REAL_TO_WORD(gUI.TiG.arrPV[6].sNum[8].rPercent);	//E16L2

gModbus.master.sPos.arrDat[218]:= REAL_TO_WORD(gUI.TiG.arrPV[7].sNum[20].rPercent);	//E17L1
gModbus.master.sPos.arrDat[219]:= REAL_TO_WORD(gUI.TiG.arrPV[7].sNum[21].rPercent);	//E17L2
gModbus.master.sPos.arrDat[220]:= REAL_TO_WORD(gUI.TiG.arrPV[7].sNum[1].rPercent);	//E18L
gModbus.master.sPos.arrDat[221]:= REAL_TO_WORD(gUI.TiG.arrPV[7].sNum[2].rPercent);	//E19L
gModbus.master.sPos.arrDat[222]:= REAL_TO_WORD(gUI.TiG.arrPV[7].sNum[3].rPercent);	//E20L
gModbus.master.sPos.arrDat[223]:= REAL_TO_WORD(gUI.TiG.arrPV[7].sNum[4].rPercent);	
gModbus.master.sPos.arrDat[224]:= REAL_TO_WORD(gUI.TiG.arrPV[7].sNum[5].rPercent);
gModbus.master.sPos.arrDat[225]:= REAL_TO_WORD(gUI.TiG.arrPV[7].sNum[6].rPercent);
gModbus.master.sPos.arrDat[226]:= REAL_TO_WORD(gUI.TiG.arrPV[7].sNum[7].rPercent);
gModbus.master.sPos.arrDat[227]:= REAL_TO_WORD(gUI.TiG.arrPV[7].sNum[8].rPercent);
gModbus.master.sPos.arrDat[228]:= REAL_TO_WORD(gUI.TiG.arrPV[7].sNum[9].rPercent);	//E26L
gModbus.master.sPos.arrDat[229]:= REAL_TO_WORD(gUI.TiG.arrPV[7].sNum[22].rPercent);	//E27L1
gModbus.master.sPos.arrDat[230]:= REAL_TO_WORD(gUI.TiG.arrPV[7].sNum[23].rPercent);	//E27L2

gModbus.master.sPos.arrDat[231]:= REAL_TO_WORD(gUI.TiG.arrPV[1].sNum[1].rPercent);	//E28L1
gModbus.master.sPos.arrDat[232]:= REAL_TO_WORD(gUI.TiG.arrPV[1].sNum[2].rPercent);	//E28L2
gModbus.master.sPos.arrDat[233]:= REAL_TO_WORD(gUI.TiG.arrPV[1].sNum[3].rPercent);	//E29L
gModbus.master.sPos.arrDat[234]:= REAL_TO_WORD(gUI.TiG.arrPV[1].sNum[4].rPercent);	//E30L

FOR iTemp:=0 TO 7 DO
	gModbus.master.sPos.arrDat[235+iTemp]:= REAL_TO_WORD(gUI.TiG.arrPV[3].sNum[1+iTemp].rPercent);
	gModbus.master.sPos.arrDat[243+iTemp]:= REAL_TO_WORD(gUI.TiG.arrPV[4].sNum[1+iTemp].rPercent);
	gModbus.master.sPos.arrDat[251+iTemp]:= REAL_TO_WORD(gUI.TiG.arrPV[4].sNum[1+iTemp].rPercent);
END_FOR

gModbus.master.sPos.arrDat[259]:= REAL_TO_WORD(gUI.TiG.arrPV[6].sNum[1].rPercent);	//E13Q
gModbus.master.sPos.arrDat[260]:= REAL_TO_WORD(gUI.TiG.arrPV[6].sNum[2].rPercent);	//E14Q
gModbus.master.sPos.arrDat[261]:= REAL_TO_WORD(gUI.TiG.arrPV[6].sNum[3].rPercent);	//E15Q没有16Q

FOR iTemp:=0 TO 9 DO
gModbus.master.sPos.arrDat[262+iTemp]:= REAL_TO_WORD(gUI.TiG.arrPV[7].sNum[10+iTemp].rPercent);//E17Q-E26Q
END_FOR

gModbus.master.sPos.arrDat[272]:= REAL_TO_WORD(gUI.TiG.arrPV[1].sNum[10].rPercent);	//E28Q
gModbus.master.sPos.arrDat[273]:= REAL_TO_WORD(gUI.TiG.arrPV[1].sNum[11].rPercent);	//E29Q
gModbus.master.sPos.arrDat[274]:= REAL_TO_WORD(gUI.TiG.arrPV[1].sNum[12].rPercent);	//E30Q
END_METHOD

METHOD PRIVATE executeCmd0
VAR_INPUT
	
END_VAR
VAR 

	arrExecute	:ARRAY [20..23,0..15] OF BOOL;
	iTemp1		:USINT;
	iTemp2		:USINT;
	bToken		:BOOL;
	i2H			:USINT;//iTemp2Half:=iTemp2/2
END_VAR
VAR CONSTANT
	a0PV		:ARRAY [0..7] OF USINT :=[1,1,2,2,2,2,2,6];	
	a0PV1		:ARRAY [0..7] OF USINT :=[3,6,1,2,3,4,5,4];		
	a1PV		:ARRAY [0..7] OF USINT :=[6,6,7,7,7,7,7,1];	
	a1PV1		:ARRAY [0..7] OF USINT :=[3,5,6,1,2,3,7,1];	
	a2PV		:ARRAY [0..7] OF USINT :=[1,3,4,5,6,6,7,7];	
	a2PV1		:ARRAY [0..7] OF USINT :=[2,1,1,1,1,2,4,5];		
	a3PV		:ARRAY [0..7] OF USINT :=[1,1];	
	a3PV1		:ARRAY [0..7] OF USINT :=[5,4];	
END_VAR
FOR iTemp:=20 TO 23 DO
	gModbus.master.sCmd.arrNew[iTemp,0]:=gModbus.master.sCmd.arrDat[iTemp].0;
	gModbus.master.sCmd.arrNew[iTemp,1]:=gModbus.master.sCmd.arrDat[iTemp].1;
	gModbus.master.sCmd.arrNew[iTemp,2]:=gModbus.master.sCmd.arrDat[iTemp].2;
	gModbus.master.sCmd.arrNew[iTemp,3]:=gModbus.master.sCmd.arrDat[iTemp].3;
	gModbus.master.sCmd.arrNew[iTemp,4]:=gModbus.master.sCmd.arrDat[iTemp].4;
	gModbus.master.sCmd.arrNew[iTemp,5]:=gModbus.master.sCmd.arrDat[iTemp].5;
	gModbus.master.sCmd.arrNew[iTemp,6]:=gModbus.master.sCmd.arrDat[iTemp].6;
	gModbus.master.sCmd.arrNew[iTemp,7]:=gModbus.master.sCmd.arrDat[iTemp].7;
	gModbus.master.sCmd.arrNew[iTemp,8]:=gModbus.master.sCmd.arrDat[iTemp].8;
	gModbus.master.sCmd.arrNew[iTemp,9]:=gModbus.master.sCmd.arrDat[iTemp].9;
	gModbus.master.sCmd.arrNew[iTemp,10]:=gModbus.master.sCmd.arrDat[iTemp].10;
	gModbus.master.sCmd.arrNew[iTemp,11]:=gModbus.master.sCmd.arrDat[iTemp].11;
	gModbus.master.sCmd.arrNew[iTemp,12]:=gModbus.master.sCmd.arrDat[iTemp].12;
	gModbus.master.sCmd.arrNew[iTemp,13]:=gModbus.master.sCmd.arrDat[iTemp].13;
	gModbus.master.sCmd.arrNew[iTemp,14]:=gModbus.master.sCmd.arrDat[iTemp].14;
	gModbus.master.sCmd.arrNew[iTemp,15]:=gModbus.master.sCmd.arrDat[iTemp].15;
END_FOR

FOR iTemp1:=20 TO 23 DO
	FOR iTemp2:=0 TO 15 DO
		IF gModbus.master.sCmd.arrNew[iTemp1,iTemp2]>gModbus.master.sCmd.arrLast[iTemp1,iTemp2] THEN
			i2H:=iTemp2/2;
			IF (iTemp2 MOD 2) = 0 THEN	//伸出
				CASE iTemp1 OF
				20:gUI.TiG.arrPV[a0PV[i2H]].sColumn[a0PV1[i2H]].bExtend:=TRUE;
				21:gUI.TiG.arrPV[a1PV[i2H]].sColumn[a1PV1[i2H]].bExtend:=TRUE;
				22:gUI.TiG.arrPV[a2PV[i2H]].sColumn[a2PV1[i2H]].bExtend:=TRUE;
				23:gUI.TiG.arrPV[a3PV[i2H]].sColumn[a3PV1[i2H]].bExtend:=TRUE;
				END_CASE
			ELSE						//缩回
				CASE iTemp1 OF
				20:gUI.TiG.arrPV[a0PV[i2H]].sColumn[a0PV1[i2H]].bRetract:=TRUE;
				21:gUI.TiG.arrPV[a1PV[i2H]].sColumn[a1PV1[i2H]].bRetract:=TRUE;
				22:gUI.TiG.arrPV[a2PV[i2H]].sColumn[a2PV1[i2H]].bRetract:=TRUE;
				23:gUI.TiG.arrPV[a3PV[i2H]].sColumn[a3PV1[i2H]].bRetract:=TRUE;
				END_CASE
			END_IF
			//bToken:=TRUE;	//有上升沿则记录
			//arrExecute[iTemp1,iTemp2]:=1;
			
			
		END_IF
		gModbus.master.sCmd.arrLast[iTemp1,iTemp2]:=gModbus.master.sCmd.arrNew[iTemp1,iTemp2];
	END_FOR
END_FOR



